(* CODESYS project SmiuUGP_Dubniki.project

Project tree, tasks and I/O mapping:
  CODESYS_Control_for_Raspberry_Pi : CODESYS Control for Raspberry Pi, 3S - Smart Software Solutions GmbH, version 3.5.7.10
    application Application
      libraries: Util, * (System); AlarmManager, * (Intern); Alarm Manager Interfaces, * (Intern); Standard, * (System); VisuDialogs, * (System)
      task MainTask (cyclic, interval t#50ms, priority 2, watchdog t#1000ms x 1) calls PLC_PRG, GPIO_HANDLER, AlarmChecker
      task VISU_TASK (cyclic, interval 100 ms, priority 30) calls VisuElems.Visu_Prg
      task AlarmManagerTask (cyclic, interval 50 ms, priority 31) calls AlarmManager.Alarm_Prg
      task BusTask (cyclic, interval t#20ms, priority 1, watchdog t#1000ms x 1) calls BusReinit
      program PLC_PRG [ST]
      image pool ImagePool
      program GPIO_HANDLER [ST]
      visualization/
        visualisation monitoring
        ups_s2/
          visualisation ups_s2_state
          visualisation ups_s2_params
        visualisation main
        visualisation info
        visualisation climate
        visualisation alarm
        visualisation schrps
        visualisation shasn
        visualisation logs
        visualisation schrpa
        ups_s1/
          visualisation ups_s1_params
          visualisation ups_s1_state
        ups_a1/
          visualisation ups_a1_params
          visualisation ups_a1_state
        ups_a2/
          visualisation ups_a2_params
          visualisation ups_a2_state
        visualisation climate_log
        visualisation more
      Alarm Configuration
        alarm class Error (priority 10, acknowledge REP)
        alarm class Warning (priority 30, acknowledge REP)
        alarm class Info (priority 100, acknowledge REP)
        AlarmStorage
        text list AlarmGroup
        alarm group AlarmGroup
            1 [Error]: Comparison Equal, ExpressionToCompare TRUE, Expression AlarmChecker.shrpa_in_2_alarm - "Отсутствует напряжение на резервном вводе ЩРПА"
            2 [Error]: Comparison Equal, ExpressionToCompare FALSE, Expression GPIO_HANDLER.IN_4 - "Отсутствует напряжение на основном вводе ШАСН"
            3 [Error]: Comparison Equal, ExpressionToCompare FALSE, Expression GPIO_HANDLER.IN_5 - "Отсутствует напряжение на резервном вводе ШАСН"
            4 [Error]: Comparison Equal, ExpressionToCompare FALSE, Expression PLC_PRG.shrps_ups_bus_1 - "Отсутствует напряжение на ГП 1 ЩРПС"
            5 [Error]: Comparison Equal, ExpressionToCompare FALSE, Expression PLC_PRG.shrps_ups_bus_2 - "Отсутствует напряжение на ГП 2 ЩРПС"
            96 [Error]: Comparison Equal, ExpressionToCompare TRUE, Expression GPIO_HANDLER.IN_2 - "Пожар"
            92 [Error]: Comparison Equal, ExpressionToCompare TRUE, Expression AlarmChecker.ups_s1_out_v_alarm - "Отсутствует напряжение на выходе ИБП С1"
            45 [Error]: Comparison Equal, ExpressionToCompare TRUE, Expression PLC_PRG.mpx_a1_1_alarm - "Авария ИБП А1"
            53 [Error]: Comparison Equal, ExpressionToCompare TRUE, Expression PLC_PRG.mpx_s2_1_alarm - "Авария ИБП С2"
            49 [Error]: Comparison Equal, ExpressionToCompare TRUE, Expression PLC_PRG.mpx_s1_1_alarm - "Авария ИБП С1"
            6 [Error]: Comparison Equal, ExpressionToCompare FALSE, Expression GPIO_HANDLER.IN_6 - "Отсутствует напряжение на шине БП ШАСН"
            97 [Error]: Comparison Equal, ExpressionToCompare TRUE, Expression GPIO_HANDLER.IN_1 - "Нарушение ШОС"
            93 [Error]: Comparison Equal, ExpressionToCompare TRUE, Expression AlarmChecker.ups_s2_out_v_alarm - "Отсутствует напряжение на выходе ИБП С2"
            101 [Error]: Comparison Equal, ExpressionToCompare TRUE, Expression AlarmChecker.shrps_in_2_alarm - "Отсутствует напряжение на резервном вводе ЩРПС"
            0 [Error]: Comparison Equal, ExpressionToCompare TRUE, Expression AlarmChecker.shrpa_in_1_alarm - "Отсутствует напряжение на основном вводе ЩРПА"
            47 [Error]: Comparison Equal, ExpressionToCompare TRUE, Expression PLC_PRG.mpx_a2_1_alarm - "Авария ИБП А2"
            94 [Error]: Comparison Equal, ExpressionToCompare TRUE, Expression AlarmChecker.ups_a1_out_v_alarm - "Отсутствует напряжение на выходе ИБП А1"
            90 [Error]: Comparison Equal, ExpressionToCompare TRUE, Expression AlarmChecker.ups_a1_in_v_alarm - "Отсутствует напряжение на входе ИБП А1"
            88 [Error]: Comparison Equal, ExpressionToCompare TRUE, Expression AlarmChecker.ups_s1_in_v_alarm - "Отсутствует напряжение на входе ИБП С1"
            98 [Error]: Comparison Equal, ExpressionToCompare TRUE, Expression GPIO_HANDLER.IN_3 - "Авария ШОС"
            100 [Error]: Comparison Equal, ExpressionToCompare TRUE, Expression AlarmChecker.shrps_in_1_alarm - "Отсутствует напряжение на основном вводе ЩРПC"
            89 [Error]: Comparison Equal, ExpressionToCompare TRUE, Expression AlarmChecker.ups_s2_in_v_alarm - "Отсутствует напряжение на входе ИБП С2"
            95 [Error]: Comparison Equal, ExpressionToCompare TRUE, Expression AlarmChecker.ups_a2_out_v_alarm - "Отсутствует напряжение на выходе ИБП А2"
            91 [Error]: Comparison Equal, ExpressionToCompare TRUE, Expression AlarmChecker.ups_a2_in_v_alarm - "Отсутствует напряжение на входе ИБП А2"
            7 [Error]: Comparison Equal, ExpressionToCompare FALSE, Expression GPIO_HANDLER.IN_7 - "Отсутствует напряжение на шине ГП ШАСН"
            99 [Error]: Comparison Equal, ExpressionToCompare TRUE, Expression AlarmChecker.shrpa_out_alarm - "Отсутствует напряжение на ШБПА  ЩРПА"
        text list ClimateGroup
        alarm group ClimateGroup
            1 [Info]: Comparison Equal, ExpressionToCompare TRUE, Expression PLC_PRG.climate_auto_state - "Автоматика включена"
            2 [Info]: Comparison Equal, ExpressionToCompare FALSE, Expression PLC_PRG.climate_heat_state - "Обогрев выключен"
            3 [Info]: Comparison Equal, ExpressionToCompare FALSE, Expression PLC_PRG.climate_auto_state - "Автоматика выключена"
            4 [Info]: Comparison Equal, ExpressionToCompare TRUE, Expression PLC_PRG.climate_zaslonka_state - "Заслонка открыта"
            5 [Info]: Comparison Equal, ExpressionToCompare FALSE, Expression PLC_PRG.climate_zaslonka_state - "Заслонка закрыта"
            11 [Info]: Comparison Equal, ExpressionToCompare FALSE, Expression PLC_PRG.climate_heat_door_state - "Обогрев дверей выключен"
            7 [Info]: Comparison Equal, ExpressionToCompare FALSE, Expression PLC_PRG.climate_vent_1_state - "Вентиляторы выключены"
            6 [Info]: Comparison Equal, ExpressionToCompare TRUE, Expression PLC_PRG.climate_vent_1_state - "Вентиляторы включены"
            12 [Info]: Comparison Equal, ExpressionToCompare TRUE, Expression PLC_PRG.climate_temp_low - "Низкая температура"
            13 [Info]: Comparison Equal, ExpressionToCompare TRUE, Expression PLC_PRG.climate_temp_hight - "Высокая температура"
            8 [Info]: Comparison Equal, ExpressionToCompare TRUE, Expression PLC_PRG.climate_condition_1_state - "Кондиционеры включены"
            9 [Info]: Comparison Equal, ExpressionToCompare FALSE, Expression PLC_PRG.climate_condition_1_state - "Кондиционеры выключены"
            10 [Info]: Comparison Equal, ExpressionToCompare TRUE, Expression PLC_PRG.climate_heat_door_state - "Обогрев дверей включен"
            0 [Info]: Comparison Equal, ExpressionToCompare TRUE, Expression PLC_PRG.climate_heat_state - "Обогрев включен"
      program BusReinit [ST]
      program AlarmChecker [ST]
    SoftMotion General Axis Pool
    GPIOs_B_Pi2 : GPIOs B+/Pi2, 3S - Smart Software Solutions GmbH, version 1.1.1.10
        input  Application.GPIO_HANDLER.RAW_IN_10 : BOOL  // digital inputs (GPIO0..GPIO31).Bit5
        input  Application.GPIO_HANDLER.RAW_IN_12 : BOOL  // digital inputs (GPIO0..GPIO31).Bit6
        input  Application.GPIO_HANDLER.RAW_IN_9 : BOOL  // digital inputs (GPIO0..GPIO31).Bit7
        input  Application.GPIO_HANDLER.RAW_IN_8 : BOOL  // digital inputs (GPIO0..GPIO31).Bit8
        input  Application.GPIO_HANDLER.RAW_IN_3 : BOOL  // digital inputs (GPIO0..GPIO31).Bit10
        input  Application.GPIO_HANDLER.RAW_IN_11 : BOOL  // digital inputs (GPIO0..GPIO31).Bit12
        input  Application.GPIO_HANDLER.RAW_IN_1 : BOOL  // digital inputs (GPIO0..GPIO31).Bit13
        input  Application.GPIO_HANDLER.RAW_IN_6 : BOOL  // digital inputs (GPIO0..GPIO31).Bit18
        input  Application.GPIO_HANDLER.RAW_IN_7 : BOOL  // digital inputs (GPIO0..GPIO31).Bit21
        input  Application.GPIO_HANDLER.RAW_IN_5 : BOOL  // digital inputs (GPIO0..GPIO31).Bit23
        input  Application.GPIO_HANDLER.RAW_IN_4 : BOOL  // digital inputs (GPIO0..GPIO31).Bit24
        input  Application.GPIO_HANDLER.RAW_IN_2 : BOOL  // digital inputs (GPIO0..GPIO31).Bit25
        unmapped channels: digital inputs (GPIO0..GPIO31), digital outputs (GPIO0..GPIO31)
    Camera device
      <Empty>
    I²C
    SPI
    Onewire
    Ethernet : Ethernet, 3S - Smart Software Solutions GmbH, version 3.4.2.0
        settings: IPAddress = [192,168,10,200]; SubnetMask = [255,255,255,0]; GatewayAddress = [0,0,0,0]; NetworkInterfaceName = 'eth0'; NetworkInterfaceName = "eth0"
      Modbus_TCP_Master : Modbus TCP Master, 3S - Smart Software Solutions GmbH, version 3.5.4.0
          settings: AutoReconnect = TRUE
        IPS_2_2 : Modbus TCP Slave, 3S - Smart Software Solutions GmbH, version 3.5.4.0
            settings: Unit-ID = 1; ResponseTimeout = 1500; IPAddress = [192, 168, 10, 204]; Input_group.Function Code = 3; Input_group.Read Offset = 16#006D; Input_group.Read Length = 4; Input_group.Write Offset = 0; Input_group.Write Length = 0; Input_group.Cycle Time = 300; Output_group.Function Code = 3; Output_group.Read Offset = 16#0077; Output_group.Read Length = 7; Output_group.Write Offset = 0; Output_group.Write Length = 0; Output_group.Cycle Time = 300; Bypass_group.Function Code = 3; Bypass_group.Read Offset = 16#0081; Bypass_group.Read Length = 4; Bypass_group.Write Offset = 0; Bypass_group.Write Length = 0; Bypass_group.Cycle Time = 300; Battarey_group.Function Code = 3; Battarey_group.Read Offset = 16#0063; Battarey_group.Read Length = 4; Battarey_group.Write Offset = 0; Battarey_group.Write Length = 0; Battarey_group.Cycle Time = 300; Inv_Byp.Function Code = 3; Inv_Byp.Read Offset = 16#0095; Inv_Byp.Read Length = 1; Inv_Byp.Write Offset = 0; Inv_Byp.Write Length = 0; Inv_Byp.Cycle Time = 300; Status_group2.Function Code = 3; Status_group2.Read Offset = 16#0031; Status_group2.Read Length = 4; Status_group2.Write Offset = 0; Status_group2.Write Length = 0; Status_group2.Cycle Time = 300; Ivertor.Function Code = 3;
              Ivertor.Read Offset = 16#0096; Ivertor.Read Length = 1; Ivertor.Write Offset = 0; Ivertor.Write Length = 0; Ivertor.Cycle Time = 300; Battarey_temp.Function Code = 3; Battarey_temp.Read Offset = 16#001D; Battarey_temp.Read Length = 1; Battarey_temp.Write Offset = 0; Battarey_temp.Write Length = 0; Battarey_temp.Cycle Time = 300; Fault_grup.Function Code = 3; Fault_grup.Read Offset = 16#009F; Fault_grup.Read Length = 7; Fault_grup.Write Offset = 0; Fault_grup.Write Length = 0; Fault_grup.Cycle Time = 300
            input  Application.PLC_PRG.mpx_s2_1_in_freq : WORD  // Input_group.Input_group
            input  Application.PLC_PRG.mpx_s2_1_in_v_1 : WORD  // Input_group.Input_group
            input  Application.PLC_PRG.mpx_s2_1_in_v_2 : WORD  // Input_group.Input_group
            input  Application.PLC_PRG.mpx_s2_1_in_v_3 : WORD  // Input_group.Input_group
            input  Application.PLC_PRG.mpx_s2_1_output_freq : WORD  // Output_group.Output_group
            input  Application.PLC_PRG.mpx_s2_1_output_v_1 : WORD  // Output_group.Output_group
            input  Application.PLC_PRG.mpx_s2_1_output_v_2 : WORD  // Output_group.Output_group
            input  Application.PLC_PRG.mpx_s2_1_output_v_3 : WORD  // Output_group.Output_group
            input  Application.PLC_PRG.mpx_s2_1_load_ph_1 : WORD  // Output_group.Output_group
            input  Application.PLC_PRG.mpx_s2_1_load_ph_2 : WORD  // Output_group.Output_group
            input  Application.PLC_PRG.mpx_s2_1_load_ph_3 : WORD  // Output_group.Output_group
            input  Application.PLC_PRG.mpx_s2_1_bypass_freq : WORD  // Bypass_group.Bypass_group
            input  Application.PLC_PRG.mpx_s2_1_bypass_v_1 : WORD  // Bypass_group.Bypass_group
            input  Application.PLC_PRG.mpx_s2_1_bypass_v_2 : WORD  // Bypass_group.Bypass_group
            input  Application.PLC_PRG.mpx_s2_1_bypass_v_3 : WORD  // Bypass_group.Bypass_group
            input  Application.PLC_PRG.mpx_s2_1_battery_voltage : WORD  // Battarey_group.Battarey_group
            input  Application.PLC_PRG.mpx_s2_1_battery_capacity : WORD  // Battarey_group.Battarey_group
            input  Application.PLC_PRG.mpx_s2_time_m : WORD  // Battarey_group.Battarey_group
            input  Application.PLC_PRG.mpx_s2_1_battery_current : WORD  // Battarey_group.Battarey_group
            input  Application.PLC_PRG.mpx_s2_1_inv_byp : ARRAY[0..0] OF WORD  // Inv_Byp
            input  Application.PLC_PRG.mpx_s2_1_state_reg : WORD  // Status_group2.Status_group2
            input  Application.PLC_PRG.mpx_s2_1_Invertor : ARRAY[0..0] OF WORD  // Ivertor
            input  Application.PLC_PRG.mpx_s2_1_temp : ARRAY[0..0] OF WORD  // Battarey_temp
            input  Application.PLC_PRG.mpx_s2_1_emergency : WORD  // Fault_grup.Fault_grup
            input  Application.PLC_PRG.mpx_s2_1_overload : WORD  // Fault_grup.Fault_grup
            input  Application.PLC_PRG.mpx_s2_1_outfail : WORD  // Fault_grup.Fault_grup
            input  Application.PLC_PRG.mpx_s2_1_overtemp : WORD  // Fault_grup.Fault_grup
            unmapped channels: Input_group, Output_group, Bypass_group, Battarey_group, Status_group2, Fault_grup
        IPS_2_1 : Modbus TCP Slave, 3S - Smart Software Solutions GmbH, version 3.5.4.0
            settings: Unit-ID = 1; ResponseTimeout = 1500; IPAddress = [192, 168, 10, 203]; Input_group.Function Code = 3; Input_group.Read Offset = 16#006D; Input_group.Read Length = 4; Input_group.Write Offset = 0; Input_group.Write Length = 0; Input_group.Cycle Time = 300; Output_group.Function Code = 3; Output_group.Read Offset = 16#0077; Output_group.Read Length = 7; Output_group.Write Offset = 0; Output_group.Write Length = 0; Output_group.Cycle Time = 300; Bypass_group.Function Code = 3; Bypass_group.Read Offset = 16#0081; Bypass_group.Read Length = 4; Bypass_group.Write Offset = 0; Bypass_group.Write Length = 0; Bypass_group.Cycle Time = 300; Battarey_group.Function Code = 3; Battarey_group.Read Offset = 16#0063; Battarey_group.Read Length = 4; Battarey_group.Write Offset = 0; Battarey_group.Write Length = 0; Battarey_group.Cycle Time = 300; Status2_group.Function Code = 3; Status2_group.Read Offset = 16#0031; Status2_group.Read Length = 4; Status2_group.Write Offset = 0; Status2_group.Write Length = 0; Status2_group.Cycle Time = 300; Invertor.Function Code = 3; Invertor.Read Offset = 16#0096; Invertor.Read Length = 1; Invertor.Write Offset = 0; Invertor.Write Length = 0; Invertor.Cycle Time = 300; Battarey_temp.Function Code = 3;
              Battarey_temp.Read Offset = 16#001D; Battarey_temp.Read Length = 1; Battarey_temp.Write Offset = 0; Battarey_temp.Write Length = 0; Battarey_temp.Cycle Time = 300; Inv_Byp.Function Code = 3; Inv_Byp.Read Offset = 16#0095; Inv_Byp.Read Length = 1; Inv_Byp.Write Offset = 0; Inv_Byp.Write Length = 0; Inv_Byp.Cycle Time = 300; Fault_group.Function Code = 3; Fault_group.Read Offset = 16#009F; Fault_group.Read Length = 7; Fault_group.Write Offset = 0; Fault_group.Write Length = 0; Fault_group.Cycle Time = 300
            input  Application.PLC_PRG.mpx_s1_1_in_freq : WORD  // Input_group.Input_group
            input  Application.PLC_PRG.mpx_s1_1_in_v_1 : WORD  // Input_group.Input_group
            input  Application.PLC_PRG.mpx_s1_1_in_v_2 : WORD  // Input_group.Input_group
            input  Application.PLC_PRG.mpx_s1_1_in_v_3 : WORD  // Input_group.Input_group
            input  Application.PLC_PRG.mpx_s1_1_output_freq : WORD  // Output_group.Output_group
            input  Application.PLC_PRG.mpx_s1_1_output_v_1 : WORD  // Output_group.Output_group
            input  Application.PLC_PRG.mpx_s1_1_output_v_2 : WORD  // Output_group.Output_group
            input  Application.PLC_PRG.mpx_s1_1_output_v_3 : WORD  // Output_group.Output_group
            input  Application.PLC_PRG.mpx_s1_1_load_ph_1 : WORD  // Output_group.Output_group
            input  Application.PLC_PRG.mpx_s1_1_load_ph_2 : WORD  // Output_group.Output_group
            input  Application.PLC_PRG.mpx_s1_1_load_ph_3 : WORD  // Output_group.Output_group
            input  Application.PLC_PRG.mpx_s1_1_bypass_freq : WORD  // Bypass_group.Bypass_group
            input  Application.PLC_PRG.mpx_s1_1_bypass_v_1 : WORD  // Bypass_group.Bypass_group
            input  Application.PLC_PRG.mpx_s1_1_bypass_v_2 : WORD  // Bypass_group.Bypass_group
            input  Application.PLC_PRG.mpx_s1_1_bypass_v_3 : WORD  // Bypass_group.Bypass_group
            input  Application.PLC_PRG.mpx_s1_1_battery_voltage : WORD  // Battarey_group.Battarey_group
            input  Application.PLC_PRG.mpx_s1_1_battery_capacity : WORD  // Battarey_group.Battarey_group
            input  Application.PLC_PRG.mpx_s1_time_m : WORD  // Battarey_group.Battarey_group
            input  Application.PLC_PRG.mpx_s1_1_battery_current : WORD  // Battarey_group.Battarey_group
            input  Application.PLC_PRG.mpx_s1_1_state_reg : WORD  // Status2_group.Status2_group
            input  Application.PLC_PRG.mpx_s1_1_Invertor : ARRAY[0..0] OF WORD  // Invertor
            input  Application.PLC_PRG.mpx_s1_1_temp : ARRAY[0..0] OF WORD  // Battarey_temp
            input  Application.PLC_PRG.mpx_s1_1_inv_byp : ARRAY[0..0] OF WORD  // Inv_Byp
            input  Application.PLC_PRG.mpx_s1_1_emergency : WORD  // Fault_group.Fault_group
            input  Application.PLC_PRG.mpx_s1_1_overload : WORD  // Fault_group.Fault_group
            input  Application.PLC_PRG.mpx_s1_1_outfail : WORD  // Fault_group.Fault_group
            input  Application.PLC_PRG.mpx_s1_1_overtemp : WORD  // Fault_group.Fault_group
            unmapped channels: Input_group, Output_group, Bypass_group, Battarey_group, Status2_group, Fault_group
        IPS_1_1 : Modbus TCP Slave, 3S - Smart Software Solutions GmbH, version 3.5.4.0
            settings: Unit-ID = 1; ResponseTimeout = 1500; IPAddress = [192, 168, 10, 201]; Input_group.Function Code = 3; Input_group.Read Offset = 16#006D; Input_group.Read Length = 4; Input_group.Write Offset = 0; Input_group.Write Length = 0; Input_group.Cycle Time = 300; Output_group.Function Code = 3; Output_group.Read Offset = 16#0077; Output_group.Read Length = 5; Output_group.Write Offset = 0; Output_group.Write Length = 0; Output_group.Cycle Time = 300; Bypass_group.Function Code = 3; Bypass_group.Read Offset = 16#0081; Bypass_group.Read Length = 2; Bypass_group.Write Offset = 0; Bypass_group.Write Length = 0; Bypass_group.Cycle Time = 300; Battarey_group.Function Code = 3; Battarey_group.Read Offset = 16#0063; Battarey_group.Read Length = 4; Battarey_group.Write Offset = 0; Battarey_group.Write Length = 0; Battarey_group.Cycle Time = 300; Status_group2.Function Code = 3; Status_group2.Read Offset = 16#0031; Status_group2.Read Length = 4; Status_group2.Write Offset = 0; Status_group2.Write Length = 0; Status_group2.Cycle Time = 300; Invertor.Function Code = 3; Invertor.Read Offset = 16#0096; Invertor.Read Length = 1; Invertor.Write Offset = 0; Invertor.Write Length = 0; Invertor.Cycle Time = 300; Battarey_temp.Function Code = 3;
              Battarey_temp.Read Offset = 16#001D; Battarey_temp.Read Length = 1; Battarey_temp.Write Offset = 0; Battarey_temp.Write Length = 0; Battarey_temp.Cycle Time = 300; Inv_Byp.Function Code = 3; Inv_Byp.Read Offset = 16#0095; Inv_Byp.Read Length = 1; Inv_Byp.Write Offset = 0; Inv_Byp.Write Length = 0; Inv_Byp.Cycle Time = 300; Fault_group.Function Code = 3; Fault_group.Read Offset = 16#009F; Fault_group.Read Length = 7; Fault_group.Write Offset = 0; Fault_group.Write Length = 0; Fault_group.Cycle Time = 300
            input  Application.PLC_PRG.mpx_a1_1_in_freq : WORD  // Input_group.Input_group
            input  Application.PLC_PRG.mpx_a1_1_in_v_1 : WORD  // Input_group.Input_group
            input  Application.PLC_PRG.mpx_a1_1_in_v_2 : WORD  // Input_group.Input_group
            input  Application.PLC_PRG.mpx_a1_1_in_v_3 : WORD  // Input_group.Input_group
            input  Application.PLC_PRG.mpx_a1_1_output_freq : WORD  // Output_group.Output_group
            input  Application.PLC_PRG.mpx_a1_1_output_v_1 : WORD  // Output_group.Output_group
            input  Application.PLC_PRG.mpx_a1_1_load_ph_1 : WORD  // Output_group.Output_group
            input  Application.PLC_PRG.mpx_a1_1_bypass_freq : WORD  // Bypass_group.Bypass_group
            input  Application.PLC_PRG.mpx_a1_1_bypass_v_1 : WORD  // Bypass_group.Bypass_group
            input  Application.PLC_PRG.mpx_a1_1_battery_voltage : WORD  // Battarey_group.Battarey_group
            input  Application.PLC_PRG.mpx_a1_1_battery_capacity : WORD  // Battarey_group.Battarey_group
            input  Application.PLC_PRG.mpx_a1_time_m : WORD  // Battarey_group.Battarey_group
            input  Application.PLC_PRG.mpx_a1_1_battery_current : WORD  // Battarey_group.Battarey_group
            input  Application.PLC_PRG.mpx_a1_1_state_reg : WORD  // Status_group2.Status_group2
            input  Application.PLC_PRG.mpx_a1_1_Invertor : ARRAY[0..0] OF WORD  // Invertor
            input  Application.PLC_PRG.mpx_a1_1_temp : ARRAY[0..0] OF WORD  // Battarey_temp
            input  Application.PLC_PRG.mpx_a1_1_inv_byp : ARRAY[0..0] OF WORD  // Inv_Byp
            input  Application.PLC_PRG.mpx_a1_1_emergency : WORD  // Fault_group.Fault_group
            input  Application.PLC_PRG.mpx_a1_1_overload : WORD  // Fault_group.Fault_group
            input  Application.PLC_PRG.mpx_a1_1_outfail : WORD  // Fault_group.Fault_group
            input  Application.PLC_PRG.mpx_a1_1_overtemp : WORD  // Fault_group.Fault_group
            unmapped channels: Input_group, Output_group, Bypass_group, Battarey_group, Status_group2, Fault_group
        IPS_1_2 : Modbus TCP Slave, 3S - Smart Software Solutions GmbH, version 3.5.4.0
            settings: Unit-ID = 1; ResponseTimeout = 1500; IPAddress = [192, 168, 10, 202]; Input_group.Function Code = 3; Input_group.Read Offset = 16#006D; Input_group.Read Length = 4; Input_group.Write Offset = 0; Input_group.Write Length = 0; Input_group.Cycle Time = 300; Output_group.Function Code = 3; Output_group.Read Offset = 16#0077; Output_group.Read Length = 5; Output_group.Write Offset = 0; Output_group.Write Length = 0; Output_group.Cycle Time = 300; Bypass_group.Function Code = 3; Bypass_group.Read Offset = 16#0081; Bypass_group.Read Length = 2; Bypass_group.Write Offset = 0; Bypass_group.Write Length = 0; Bypass_group.Cycle Time = 300; Battarey_group.Function Code = 3; Battarey_group.Read Offset = 16#0063; Battarey_group.Read Length = 4; Battarey_group.Write Offset = 0; Battarey_group.Write Length = 0; Battarey_group.Cycle Time = 300; Status_group2.Function Code = 3; Status_group2.Read Offset = 16#0031; Status_group2.Read Length = 4; Status_group2.Write Offset = 0; Status_group2.Write Length = 0; Status_group2.Cycle Time = 300; Invertor.Function Code = 3; Invertor.Read Offset = 16#0096; Invertor.Read Length = 1; Invertor.Write Offset = 0; Invertor.Write Length = 0; Invertor.Cycle Time = 300; Battarey_temp.Function Code = 3;
              Battarey_temp.Read Offset = 16#001D; Battarey_temp.Read Length = 1; Battarey_temp.Write Offset = 0; Battarey_temp.Write Length = 0; Battarey_temp.Cycle Time = 300; Inv_Byp.Function Code = 3; Inv_Byp.Read Offset = 16#0095; Inv_Byp.Read Length = 1; Inv_Byp.Write Offset = 0; Inv_Byp.Write Length = 0; Inv_Byp.Cycle Time = 300; Fault_group.Function Code = 3; Fault_group.Read Offset = 16#009F; Fault_group.Read Length = 7; Fault_group.Write Offset = 0; Fault_group.Write Length = 0; Fault_group.Cycle Time = 300
            input  Application.PLC_PRG.mpx_a2_1_in_freq : WORD  // Input_group.Input_group
            input  Application.PLC_PRG.mpx_a2_1_in_v_1 : WORD  // Input_group.Input_group
            input  Application.PLC_PRG.mpx_a2_1_in_v_2 : WORD  // Input_group.Input_group
            input  Application.PLC_PRG.mpx_a2_1_in_v_3 : WORD  // Input_group.Input_group
            input  Application.PLC_PRG.mpx_a2_1_output_freq : WORD  // Output_group.Output_group
            input  Application.PLC_PRG.mpx_a2_1_output_v_1 : WORD  // Output_group.Output_group
            input  Application.PLC_PRG.mpx_a2_1_load_ph_1 : WORD  // Output_group.Output_group
            input  Application.PLC_PRG.mpx_a2_1_bypass_freq : WORD  // Bypass_group.Bypass_group
            input  Application.PLC_PRG.mpx_a2_1_bypass_v_1 : WORD  // Bypass_group.Bypass_group
            input  Application.PLC_PRG.mpx_a2_1_battery_voltage : WORD  // Battarey_group.Battarey_group
            input  Application.PLC_PRG.mpx_a2_1_battery_capacity : WORD  // Battarey_group.Battarey_group
            input  Application.PLC_PRG.mpx_a2_time_m : WORD  // Battarey_group.Battarey_group
            input  Application.PLC_PRG.mpx_a2_1_battery_current : WORD  // Battarey_group.Battarey_group
            input  Application.PLC_PRG.mpx_a2_1_state_reg : WORD  // Status_group2.Status_group2
            input  Application.PLC_PRG.mpx_a2_1_Invertor : ARRAY[0..0] OF WORD  // Invertor
            input  Application.PLC_PRG.mpx_a2_1_temp : ARRAY[0..0] OF WORD  // Battarey_temp
            input  Application.PLC_PRG.mpx_a2_1_inv_byp : ARRAY[0..0] OF WORD  // Inv_Byp
            input  Application.PLC_PRG.mpx_a2_1_emergency : WORD  // Fault_group.Fault_group
            input  Application.PLC_PRG.mpx_a2_1_overload : WORD  // Fault_group.Fault_group
            input  Application.PLC_PRG.mpx_a2_1_outfail : WORD  // Fault_group.Fault_group
            input  Application.PLC_PRG.mpx_a2_1_overtemp : WORD  // Fault_group.Fault_group
            unmapped channels: Input_group, Output_group, Bypass_group, Battarey_group, Status_group2, Fault_group
    ModbusIN : Modbus COM, 3S - Smart Software Solutions GmbH, version 3.4.0.0
        settings: DataBits = 8; StopBits = 1; ComPort = 1
      ModbusMaster : Modbus Master, COM Port, 3S - Smart Software Solutions GmbH, version 3.5.5.0
          settings: Transmission = 'RTU'; ResponseTimeout = 60; TimeBetweenFrames = 20; Auto-restart communication = TRUE
        PLC : Modbus Slave, COM Port, 3S - Smart Software Solutions GmbH, version 3.5.4.0
            settings: SlaveAddress = 1; ResponseTimeout = 100; UseExtendedFunctionCodes = TRUE; Channel 0.Function Code = 3; Channel 0.Read Offset = 16#EB28; Channel 0.Read Length = 3; Channel 0.Write Offset = 0; Channel 0.Write Length = 0; Channel 0.Cycle Time = 500
            input  Application.PLC_PRG.climate_temp_in : WORD  // Channel 0.Channel 0
            input  Application.PLC_PRG.climate_temp_out : WORD  // Channel 0.Channel 0
            input  Application.PLC_PRG.climate_state_reg : WORD  // Channel 0.Channel 0
            unmapped channels: Channel 0
        SHRPA_ICP_CON : Modbus Slave, COM Port, 3S - Smart Software Solutions GmbH, version 3.5.4.0
            settings: SlaveAddress = 101; ResponseTimeout = 50; UseExtendedFunctionCodes = TRUE; DI.Function Code = 2; DI.Read Offset = 16#0000; DI.Read Length = 16; DI.Write Offset = 0; DI.Write Length = 0; DI.Cycle Time = 100
            input  Application.PLC_PRG.shrpa_in_1 : BOOL  // DI.DI.Bit0
            input  Application.PLC_PRG.shrpa_in_2 : BOOL  // DI.DI.Bit1
            input  Application.PLC_PRG.shrpa_ups_in_1_raw : BOOL  // DI.DI.Bit2
            input  Application.PLC_PRG.shrpa_ups_in_2_raw : BOOL  // DI.DI.Bit3
            input  Application.PLC_PRG.shrpa_input_switch_state_1 : BOOL  // DI.DI.Bit4
            input  Application.PLC_PRG.shrpa_input_switch_state_2 : BOOL  // DI.DI.Bit5
            input  Application.PLC_PRG.shrpa_ups_out_1 : BOOL  // DI.DI.Bit6
            input  Application.PLC_PRG.shrpa_ups_out_2 : BOOL  // DI.DI.Bit7
            input  Application.PLC_PRG.shrpa_load_line_1_source_state_1 : BOOL  // DI.DI.Bit0
            input  Application.PLC_PRG.shrpa_load_line_1_source_state_2 : BOOL  // DI.DI.Bit1
            input  Application.PLC_PRG.shrpa_load_line_2_source_state_2 : BOOL  // DI.DI.Bit2
            input  Application.PLC_PRG.shrpa_load_line_2_source_state_1 : BOOL  // DI.DI.Bit3
            input  Application.PLC_PRG.shrpa_input_tv1 : BOOL  // DI.DI.Bit4
            input  Application.PLC_PRG.shrpa_bypass_in_1 : BOOL  // DI.DI.Bit5
            input  Application.PLC_PRG.shrpa_bypass_in_2 : BOOL  // DI.DI.Bit6
            unmapped channels: DI
        SHRPS_ICP_CON : Modbus Slave, COM Port, 3S - Smart Software Solutions GmbH, version 3.5.4.0
            settings: SlaveAddress = 102; ResponseTimeout = 50; UseExtendedFunctionCodes = TRUE; DI.Function Code = 2; DI.Read Offset = 16#0000; DI.Read Length = 16; DI.Write Offset = 0; DI.Write Length = 0; DI.Cycle Time = 100
            input  Application.PLC_PRG.shrps_in_1 : BOOL  // DI.DI.Bit0
            input  Application.PLC_PRG.shrps_in_2 : BOOL  // DI.DI.Bit1
            input  Application.PLC_PRG.shrps_ups_in_1 : BOOL  // DI.DI.Bit2
            input  Application.PLC_PRG.shrps_bypass_in_1 : BOOL  // DI.DI.Bit3
            input  Application.PLC_PRG.shrps_ups_in_2 : BOOL  // DI.DI.Bit4
            input  Application.PLC_PRG.shrps_bypass_in_2 : BOOL  // DI.DI.Bit5
            input  Application.PLC_PRG.shrps_ups_out_1 : BOOL  // DI.DI.Bit6
            input  Application.PLC_PRG.shrps_ups_out_2 : BOOL  // DI.DI.Bit7
            input  Application.PLC_PRG.shrps_bypass_out : BOOL  // DI.DI.Bit0
            input  Application.PLC_PRG.shrps_ups_bus_1_raw : BOOL  // DI.DI.Bit1
            input  Application.PLC_PRG.shrps_ups_bus_2_raw : BOOL  // DI.DI.Bit2
            unmapped channels: DI
        SHASN_ICP_CON : Modbus Slave, COM Port, 3S - Smart Software Solutions GmbH, version 3.5.4.0
            settings: SlaveAddress = 103; ResponseTimeout = 50; UseExtendedFunctionCodes = TRUE; DI.Function Code = 2; DI.Read Offset = 16#0000; DI.Read Length = 16; DI.Write Offset = 0; DI.Write Length = 0; DI.Cycle Time = 100
            unmapped channels: DI
        SHRPA_ELNET_2 : Modbus Slave, COM Port, 3S - Smart Software Solutions GmbH, version 3.5.4.0
            settings: SlaveAddress = 12; ResponseTimeout = 100; UseExtendedFunctionCodes = TRUE; Voltage.Function Code = 3; Voltage.Read Offset = 16#0001; Voltage.Read Length = 6; Voltage.Write Offset = 0; Voltage.Write Length = 0; Voltage.Cycle Time = 500; Current.Function Code = 3; Current.Read Offset = 16#000D; Current.Read Length = 6; Current.Write Offset = 0; Current.Write Length = 0; Current.Cycle Time = 500
            input  Application.PLC_PRG.shrpa_voltage_registers2 : ARRAY[0..5] OF WORD  // Voltage
            unmapped channels: Current
        SHRPA_ELNET_1 : Modbus Slave, COM Port, 3S - Smart Software Solutions GmbH, version 3.5.4.0
            settings: SlaveAddress = 11; ResponseTimeout = 100; UseExtendedFunctionCodes = TRUE; Voltage.Function Code = 3; Voltage.Read Offset = 16#0001; Voltage.Read Length = 6; Voltage.Write Offset = 0; Voltage.Write Length = 0; Voltage.Cycle Time = 500; Current.Function Code = 3; Current.Read Offset = 16#000D; Current.Read Length = 6; Current.Write Offset = 0; Current.Write Length = 0; Current.Cycle Time = 500
            input  Application.PLC_PRG.shrpa_voltage_registers1 : ARRAY[0..5] OF WORD  // Voltage
            unmapped channels: Current
        SHRPA_ELNET_3 : Modbus Slave, COM Port, 3S - Smart Software Solutions GmbH, version 3.5.4.0
            settings: SlaveAddress = 13; ResponseTimeout = 100; UseExtendedFunctionCodes = TRUE; Voltage.Function Code = 3; Voltage.Read Offset = 16#0001; Voltage.Read Length = 2; Voltage.Write Offset = 0; Voltage.Write Length = 0; Voltage.Cycle Time = 500; Current.Function Code = 3; Current.Read Offset = 16#000D; Current.Read Length = 2; Current.Write Offset = 0; Current.Write Length = 0; Current.Cycle Time = 500; Freq.Function Code = 3; Freq.Read Offset = 16#0033; Freq.Read Length = 2; Freq.Write Offset = 0; Freq.Write Length = 0; Freq.Cycle Time = 500
            input  Application.PLC_PRG.shrpa_voltage_registers3 : ARRAY[0..1] OF WORD  // Voltage
            input  Application.PLC_PRG.shrpa_current_registers3 : ARRAY[0..1] OF WORD  // Current
            input  Application.PLC_PRG.shrpa_freq_registers3 : ARRAY[0..1] OF WORD  // Freq
        SHRPA_ELNET_4 : Modbus Slave, COM Port, 3S - Smart Software Solutions GmbH, version 3.5.4.0
            settings: SlaveAddress = 14; ResponseTimeout = 100; UseExtendedFunctionCodes = TRUE; Voltage.Function Code = 3; Voltage.Read Offset = 16#0001; Voltage.Read Length = 2; Voltage.Write Offset = 0; Voltage.Write Length = 0; Voltage.Cycle Time = 500; Current.Function Code = 3; Current.Read Offset = 16#000D; Current.Read Length = 2; Current.Write Offset = 0; Current.Write Length = 0; Current.Cycle Time = 500; Freq.Function Code = 3; Freq.Read Offset = 16#0033; Freq.Read Length = 2; Freq.Write Offset = 0; Freq.Write Length = 0; Freq.Cycle Time = 500
            input  Application.PLC_PRG.shrpa_voltage_registers4 : ARRAY[0..1] OF WORD  // Voltage
            input  Application.PLC_PRG.shrpa_current_registers4 : ARRAY[0..1] OF WORD  // Current
            input  Application.PLC_PRG.shrpa_freq_registers4 : ARRAY[0..1] OF WORD  // Freq
        SHRPS_ELNET_1 : Modbus Slave, COM Port, 3S - Smart Software Solutions GmbH, version 3.5.4.0
            settings: SlaveAddress = 21; ResponseTimeout = 100; UseExtendedFunctionCodes = TRUE; Voltage.Function Code = 3; Voltage.Read Offset = 16#0001; Voltage.Read Length = 6; Voltage.Write Offset = 0; Voltage.Write Length = 0; Voltage.Cycle Time = 500; Current.Function Code = 3; Current.Read Offset = 16#000D; Current.Read Length = 6; Current.Write Offset = 0; Current.Write Length = 0; Current.Cycle Time = 500
            input  Application.PLC_PRG.shrps_voltage_registers1 : ARRAY[0..5] OF WORD  // Voltage
            unmapped channels: Current
        SHRPS_ELNET_2 : Modbus Slave, COM Port, 3S - Smart Software Solutions GmbH, version 3.5.4.0
            settings: SlaveAddress = 22; ResponseTimeout = 100; UseExtendedFunctionCodes = TRUE; Voltage.Function Code = 3; Voltage.Read Offset = 16#0001; Voltage.Read Length = 6; Voltage.Write Offset = 0; Voltage.Write Length = 0; Voltage.Cycle Time = 500; Current.Function Code = 3; Current.Read Offset = 16#000D; Current.Read Length = 6; Current.Write Offset = 0; Current.Write Length = 0; Current.Cycle Time = 500
            input  Application.PLC_PRG.shrps_voltage_registers2 : ARRAY[0..5] OF WORD  // Voltage
            unmapped channels: Current
        SHRPS_ELNET_3 : Modbus Slave, COM Port, 3S - Smart Software Solutions GmbH, version 3.5.4.0
            settings: SlaveAddress = 23; ResponseTimeout = 100; UseExtendedFunctionCodes = TRUE; Voltage.Function Code = 3; Voltage.Read Offset = 16#0001; Voltage.Read Length = 6; Voltage.Write Offset = 0; Voltage.Write Length = 0; Voltage.Cycle Time = 500; Current.Function Code = 3; Current.Read Offset = 16#000D; Current.Read Length = 6; Current.Write Offset = 0; Current.Write Length = 0; Current.Cycle Time = 500
            input  Application.PLC_PRG.shrps_voltage_registers3 : ARRAY[0..5] OF WORD  // Voltage
            unmapped channels: Current
        SHRPS_ELNET_4 : Modbus Slave, COM Port, 3S - Smart Software Solutions GmbH, version 3.5.4.0
            settings: SlaveAddress = 24; ResponseTimeout = 100; UseExtendedFunctionCodes = TRUE; Voltage.Function Code = 3; Voltage.Read Offset = 16#0001; Voltage.Read Length = 6; Voltage.Write Offset = 0; Voltage.Write Length = 0; Voltage.Cycle Time = 500; Current.Function Code = 3; Current.Read Offset = 16#000D; Current.Read Length = 6; Current.Write Offset = 0; Current.Write Length = 0; Current.Cycle Time = 500
            input  Application.PLC_PRG.shrps_voltage_registers4 : ARRAY[0..5] OF WORD  // Voltage
            unmapped channels: Current
    ModbusOUT : Modbus COM, 3S - Smart Software Solutions GmbH, version 3.4.0.0
        settings: DataBits = 8; StopBits = 1; ComPort = 2
      Modbus_Serial_Device : Modbus Serial Device, 3S - Smart Software Solutions GmbH, version 3.5.5.0
          output Application.PLC_PRG.mpx_s1_1_battery_capacity : WORD  // Outputs.Outputs
          output Application.PLC_PRG.mpx_s1_1_battery_current : WORD  // Outputs.Outputs
          output Application.PLC_PRG.mpx_s1_1_battery_time : WORD  // Outputs.Outputs
          output Application.PLC_PRG.mpx_s1_1_battery_voltage : WORD  // Outputs.Outputs
          output Application.PLC_PRG.mpx_s1_1_bypass_v_1 : WORD  // Outputs.Outputs
          output Application.PLC_PRG.mpx_s1_1_bypass_v_2 : WORD  // Outputs.Outputs
          output Application.PLC_PRG.mpx_s1_1_bypass_v_3 : WORD  // Outputs.Outputs
          output Application.PLC_PRG.mpx_s1_1_in_v_1 : WORD  // Outputs.Outputs
          output Application.PLC_PRG.mpx_s1_1_in_v_2 : WORD  // Outputs.Outputs
          output Application.PLC_PRG.mpx_s1_1_in_v_3 : WORD  // Outputs.Outputs
          output Application.PLC_PRG.mpx_s1_1_load_ph_1 : WORD  // Outputs.Outputs
          output Application.PLC_PRG.mpx_s1_1_load_ph_2 : WORD  // Outputs.Outputs
          output Application.PLC_PRG.mpx_s1_1_load_ph_3 : WORD  // Outputs.Outputs
          output Application.PLC_PRG.mpx_s1_1_output_active_power_1 : WORD  // Outputs.Outputs
          output Application.PLC_PRG.mpx_s1_1_output_active_power_2 : WORD  // Outputs.Outputs
          output Application.PLC_PRG.mpx_s1_1_output_active_power_3 : WORD  // Outputs.Outputs
          output Application.PLC_PRG.mpx_s1_1_output_freq : WORD  // Outputs.Outputs
          output Application.PLC_PRG.mpx_s1_1_output_v_1 : WORD  // Outputs.Outputs
          output Application.PLC_PRG.mpx_s1_1_output_v_2 : WORD  // Outputs.Outputs
          output Application.PLC_PRG.mpx_s1_1_output_v_3 : WORD  // Outputs.Outputs
          output Application.PLC_PRG.mpx_s1_1_temp : WORD  // Outputs.Outputs
          output Application.PLC_PRG.ips2_1_state : WORD  // Outputs.Outputs
          output Application.PLC_PRG.mpx_s2_1_battery_capacity : WORD  // Outputs.Outputs
          output Application.PLC_PRG.mpx_s2_1_battery_current : WORD  // Outputs.Outputs
          output Application.PLC_PRG.mpx_s2_1_battery_time : WORD  // Outputs.Outputs
          output Application.PLC_PRG.mpx_s2_1_battery_voltage : WORD  // Outputs.Outputs
          output Application.PLC_PRG.mpx_s2_1_bypass_v_1 : WORD  // Outputs.Outputs
          output Application.PLC_PRG.mpx_s2_1_bypass_v_2 : WORD  // Outputs.Outputs
          output Application.PLC_PRG.mpx_s2_1_bypass_v_3 : WORD  // Outputs.Outputs
          output Application.PLC_PRG.mpx_s2_1_in_v_1 : WORD  // Outputs.Outputs
          output Application.PLC_PRG.mpx_s2_1_in_v_2 : WORD  // Outputs.Outputs
          output Application.PLC_PRG.mpx_s2_1_in_v_3 : WORD  // Outputs.Outputs
          output Application.PLC_PRG.mpx_s2_1_load_ph_1 : WORD  // Outputs.Outputs
          output Application.PLC_PRG.mpx_s2_1_load_ph_2 : WORD  // Outputs.Outputs
          output Application.PLC_PRG.mpx_s2_1_load_ph_3 : WORD  // Outputs.Outputs
          output Application.PLC_PRG.mpx_s2_1_output_active_power_1 : WORD  // Outputs.Outputs
          output Application.PLC_PRG.mpx_s2_1_output_active_power_2 : WORD  // Outputs.Outputs
          output Application.PLC_PRG.mpx_s2_1_output_active_power_3 : WORD  // Outputs.Outputs
          output Application.PLC_PRG.mpx_s2_1_output_freq : WORD  // Outputs.Outputs
          output Application.PLC_PRG.mpx_s2_1_output_v_1 : WORD  // Outputs.Outputs
          output Application.PLC_PRG.mpx_s2_1_output_v_2 : WORD  // Outputs.Outputs
          output Application.PLC_PRG.mpx_s2_1_output_v_3 : WORD  // Outputs.Outputs
          output Application.PLC_PRG.mpx_s2_1_temp : WORD  // Outputs.Outputs
          output Application.PLC_PRG.ips2_2_state : WORD  // Outputs.Outputs
          output Application.PLC_PRG.mpx_a1_1_battery_capacity : WORD  // Outputs.Outputs
          output Application.PLC_PRG.mpx_a1_1_battery_current : WORD  // Outputs.Outputs
          output Application.PLC_PRG.mpx_a1_1_battery_time : WORD  // Outputs.Outputs
          output Application.PLC_PRG.mpx_a1_1_battery_voltage : WORD  // Outputs.Outputs
          output Application.PLC_PRG.mpx_a1_1_bypass_v_1 : WORD  // Outputs.Outputs
          output Application.PLC_PRG.mpx_a1_1_in_v_1 : WORD  // Outputs.Outputs
          output Application.PLC_PRG.mpx_a1_1_in_v_2 : WORD  // Outputs.Outputs
          output Application.PLC_PRG.mpx_a1_1_in_v_3 : WORD  // Outputs.Outputs
          output Application.PLC_PRG.mpx_a1_1_load_ph_1 : WORD  // Outputs.Outputs
          output Application.PLC_PRG.mpx_a1_1_output_active_power_1 : WORD  // Outputs.Outputs
          output Application.PLC_PRG.mpx_a1_1_output_freq : WORD  // Outputs.Outputs
          output Application.PLC_PRG.mpx_a1_1_output_v_1 : WORD  // Outputs.Outputs
          output Application.PLC_PRG.mpx_a1_1_temp : WORD  // Outputs.Outputs
          output Application.PLC_PRG.ips1_1_state : WORD  // Outputs.Outputs
          output Application.PLC_PRG.mpx_a2_1_battery_capacity : WORD  // Outputs.Outputs
          output Application.PLC_PRG.mpx_a2_1_battery_current : WORD  // Outputs.Outputs
          output Application.PLC_PRG.mpx_a2_1_battery_time : WORD  // Outputs.Outputs
          output Application.PLC_PRG.mpx_a2_1_battery_voltage : WORD  // Outputs.Outputs
          output Application.PLC_PRG.mpx_a2_1_bypass_v_1 : WORD  // Outputs.Outputs
          output Application.PLC_PRG.mpx_a2_1_in_v_1 : WORD  // Outputs.Outputs
          output Application.PLC_PRG.mpx_a2_1_in_v_2 : WORD  // Outputs.Outputs
          output Application.PLC_PRG.mpx_a2_1_in_v_3 : WORD  // Outputs.Outputs
          output Application.PLC_PRG.mpx_a2_1_load_ph_1 : WORD  // Outputs.Outputs
          output Application.PLC_PRG.mpx_a2_1_output_active_power_1 : WORD  // Outputs.Outputs
          output Application.PLC_PRG.mpx_a2_1_output_freq : WORD  // Outputs.Outputs
          output Application.PLC_PRG.mpx_a2_1_output_v_1 : WORD  // Outputs.Outputs
          output Application.PLC_PRG.mpx_a2_1_temp : WORD  // Outputs.Outputs
          output Application.PLC_PRG.ips1_2_state : WORD  // Outputs.Outputs
          output Application.PLC_PRG.climate_state_reg : WORD  // Outputs.Outputs
          output Application.PLC_PRG.climate_temp_in : WORD  // Outputs.Outputs
          output Application.PLC_PRG.climate_temp_out : WORD  // Outputs.Outputs
          unmapped channels: Inputs, Outputs
  text list GlobalTextList
  5ce3da45-db07-42e7-a21c-a00fff4ed8f6|Images\bg_800.png
  5ce3da45-db07-42e7-a21c-a00fff4ed8f6|Images\mpx_state_bg.png
  5ce3da45-db07-42e7-a21c-a00fff4ed8f6|Images\ups\bypass_line_on.png
  5ce3da45-db07-42e7-a21c-a00fff4ed8f6|Images\ups\bypass_line_off.png
  5ce3da45-db07-42e7-a21c-a00fff4ed8f6|Images\ups\battery_arrow_off.png
  5ce3da45-db07-42e7-a21c-a00fff4ed8f6|Images\ups\battery_arrow_on.png
  5ce3da45-db07-42e7-a21c-a00fff4ed8f6|Images\ups\battery_line_off.png
  5ce3da45-db07-42e7-a21c-a00fff4ed8f6|Images\ups\battery_line_on.png
  5ce3da45-db07-42e7-a21c-a00fff4ed8f6|Images\ups\bypass_arrow_off.png
  5ce3da45-db07-42e7-a21c-a00fff4ed8f6|Images\ups\bypass_arrow_on.png
  5ce3da45-db07-42e7-a21c-a00fff4ed8f6|Images\ups\arrow_off.png
  5ce3da45-db07-42e7-a21c-a00fff4ed8f6|Images\ups\arrow_on.png
  5ce3da45-db07-42e7-a21c-a00fff4ed8f6|C:\workspace\SmiuUGP\Images\Proba.png
  5ce3da45-db07-42e7-a21c-a00fff4ed8f6|C:\workspace\SmiuUGP\Images\main_bg.png
  5ce3da45-db07-42e7-a21c-a00fff4ed8f6|C:\workspace\SmiuUGP\Images\bg_800.png
  5ce3da45-db07-42e7-a21c-a00fff4ed8f6|E:\YandexDisk\Скриншоты\ups.png
  5ce3da45-db07-42e7-a21c-a00fff4ed8f6|C:\workspace\SmiuUGP\Images\mpx_state_bg.png
  5ce3da45-db07-42e7-a21c-a00fff4ed8f6|C:\workspace\SmiuUGP\Images\scheme.png
  5ce3da45-db07-42e7-a21c-a00fff4ed8f6|C:\workspace\SmiuUGP\Images\more_info.png
  5ce3da45-db07-42e7-a21c-a00fff4ed8f6|C:\workspace\SmiuUGP\Images\log.png
  5ce3da45-db07-42e7-a21c-a00fff4ed8f6|C:\workspace\SmiuUGP\Images\gpio_1.png
  5ce3da45-db07-42e7-a21c-a00fff4ed8f6|release_images\schrpa.png
  5ce3da45-db07-42e7-a21c-a00fff4ed8f6|C:\workspace\SmiuUGP\Images\volt.png
  5ce3da45-db07-42e7-a21c-a00fff4ed8f6|release_images\shasn.png
  5ce3da45-db07-42e7-a21c-a00fff4ed8f6|C:\workspace\SmiuUGP\Images\battery.png
  5ce3da45-db07-42e7-a21c-a00fff4ed8f6|C:\workspace\SmiuUGP\Images\climate.png
  5ce3da45-db07-42e7-a21c-a00fff4ed8f6|C:\workspace\SmiuUGP\Images\alert.png
  5ce3da45-db07-42e7-a21c-a00fff4ed8f6|C:\workspace\SmiuUGP\Images\automation.png
  5ce3da45-db07-42e7-a21c-a00fff4ed8f6|E:\SmiuLinux\smiu_logo.png
  5ce3da45-db07-42e7-a21c-a00fff4ed8f6|C:\workspace\SmiuUGP\Images\mini_ups.png
  5ce3da45-db07-42e7-a21c-a00fff4ed8f6|release_images\shrpa.png
  5ce3da45-db07-42e7-a21c-a00fff4ed8f6|release_images\schrps.png
*)

// CODESYS_Control_for_Raspberry_Pi/Application/PLC_PRG
PROGRAM PLC_PRG
VAR	
	// Переменные для работы с ICP DAS
	// ЩРПА
	shrpa_in_1 : BOOL;							// ввод 1
	shrpa_in_2 : BOOL;							// ввод 2
	shrpa_ups_in_1_raw : BOOL;					// инвертировано
	shrpa_ups_in_2_raw : BOOL;					// инвертировано	
	shrpa_ups_in_1 : BOOL;						// ввод ИБП А1
	shrpa_ups_in_2 : BOOL;						// ввод ИБП А2
	shrpa_input_switch_state_1 : BOOL;			// QS1 в 1 положениии
	shrpa_input_switch_state_2 : BOOL;			// QS1 во 2 положениии
	shrpa_ups_out_1 : BOOL;						// выход ИБП А1
	shrpa_ups_out_2 : BOOL;						// выход ИБП А2
	shrpa_load_line_1_source_state_1 : BOOL;	//QS2 в 1 положении
	shrpa_load_line_1_source_state_2 : BOOL;	//QS2 во 2 положении
	shrpa_load_line_2_source_state_1 : BOOL;	//QS3 в 1 положении
	shrpa_load_line_2_source_state_2 : BOOL;	//QS3 во 2 положении
	shrpa_input_tv1 : BOOL	;					// ввод от TV1
	shrpa_bypass_in_1 : BOOL;					// ввод байпаса ИБП А1
	shrpa_bypass_in_2 : BOOL;					// ввод байпаса ИБП А2
	
	// ЩРПС
	shrps_in_1 : BOOL;							// ввод 1
	shrps_in_2 : BOOL;							// ввод 2
	shrps_ups_in_1 : BOOL;						// ввод ИБП C1
	shrps_ups_in_2 : BOOL;						// ввод ИБП C2		
	shrps_bypass_in_1 : BOOL;					// ввод байпаса ИБП C1
	shrps_bypass_in_2 : BOOL;					// ввод байпаса ИБП C2
	shrps_ups_out_1 : BOOL;						// выход ИБП C1
	shrps_ups_out_2 : BOOL;						// выход ИБП C2
	shrps_bypass_out : BOOL;					// 
	shrps_ups_bus_1_raw : BOOL;					// инвертировано
	shrps_ups_bus_2_raw : BOOL;					// инвертировано
	shrps_ups_bus_1 : BOOL;						// Наличие напряжения на шине бесперебойного питания 1
	shrps_ups_bus_2 : BOOL;						// Наличие напряжения на шине бесперебойного питания 2
	
	// Переменные для работы с ElNet LTE
	delay_timeout 			: TIME := T#5S;
	// ЩРПА
	shrpa_voltage_registers1: ARRAY [1..6] OF WORD;
	shrpa_voltage_registers2: ARRAY [1..6] OF WORD;
	shrpa_voltage_registers3: ARRAY [1..2] OF WORD;
	shrpa_voltage_registers4: ARRAY [1..2] OF WORD;
	
	shrpa_current_registers3: ARRAY [1..2] OF WORD;
	shrpa_current_registers4: ARRAY [1..2] OF WORD;
	
	shrpa_freq_registers3: ARRAY [1..2] OF WORD;
	shrpa_freq_registers4: ARRAY [1..2] OF WORD;
	
	Shrpa_voltage_1_delay_timer	: TON;
	Shrpa_voltage_2_delay_timer	: TON;
	Shrpa_voltage_3_delay_timer	: TON;
	Shrpa_voltage_4_delay_timer	: TON;
	
	shrpa_voltage_1_sum_checker : REAL;
	shrpa_voltage_2_sum_checker : REAL;
	
	shrpa_voltage_1_line_1 : REAL;	
	shrpa_voltage_1_line_2 : REAL;	
	shrpa_voltage_1_line_3 : REAL;	
	shrpa_voltage_2_line_1 : REAL;	
	shrpa_voltage_2_line_2 : REAL;	
	shrpa_voltage_2_line_3 : REAL;	
	shrpa_voltage_3_line_1 : REAL;	
	shrpa_voltage_4_line_1 : REAL;
	
	shrpa_current_3_line_1 : REAL;	
	shrpa_current_4_line_1 : REAL;
	
	shrpa_freq_3_line_1 : REAL;	
	shrpa_freq_4_line_1 : REAL;
	
	// ЩРПС
	shrps_voltage_registers1: ARRAY [1..6] OF WORD;
	shrps_voltage_registers2: ARRAY [1..6] OF WORD;
	shrps_voltage_registers3: ARRAY [1..6] OF WORD;
	shrps_voltage_registers4: ARRAY [1..6] OF WORD;
	
	Shrps_voltage_1_delay_timer	: TON;
	Shrps_voltage_2_delay_timer	: TON;
	Shrps_voltage_3_delay_timer	: TON;
	Shrps_voltage_4_delay_timer	: TON;
	
	shrps_voltage_1_sum_checker : REAL;
	shrps_voltage_2_sum_checker : REAL;
	shrps_voltage_3_sum_checker : REAL;
	shrps_voltage_4_sum_checker : REAL;

	shrps_voltage_1_line_1 : REAL;
	shrps_voltage_1_line_2 : REAL;
	shrps_voltage_1_line_3 : REAL;
	
	shrps_voltage_2_line_1 : REAL;
	shrps_voltage_2_line_2 : REAL;
	shrps_voltage_2_line_3 : REAL;
	
	shrps_voltage_3_line_1 : REAL;
	shrps_voltage_3_line_2 : REAL;
	shrps_voltage_3_line_3 : REAL;
	
	shrps_voltage_4_line_1 : REAL;
	shrps_voltage_4_line_2 : REAL;
	shrps_voltage_4_line_3 : REAL;


	//Визуализация
	var_true :BOOL := TRUE;
	ack		 :BOOL;
	history  :BOOL;	
	
	//Переменные для работы с климатом
	climate_temp_out          :WORD; 
	climat_temp_out_minus     :BOOL; //Бит отрицательности температуры
	climate_temp_out_real     :REAL; //Наружная температура
	climate_temp_in           :WORD; 
	climat_temp_in_minus      :BOOL; //Бит отрицательности температуры
	climate_temp_in_real      :REAL; //Внутренняя температура
	climate_state_reg         :WORD; 
	climate_state_as_bit      :WORD_AS_BIT;
	climate_zaslonka_state    :BOOL; //Состояние заслонки
	climate_vent_1_state      :BOOL; //Состояние вентилятора №1
	climate_vent_2_state      :BOOL; //Состояние вентилятора №2
	climate_condition_1_state :BOOL; //Состояние кондиционера №1
	climate_condition_2_state :BOOL; //Состояние кондиционера №2
	climate_heat_state        :BOOL; //Состояние обогрева
	climate_heat_door_state   :BOOL; //Состояние обогрева дверей
	climate_auto_state        :BOOL; //Состояние автоматики климата
	climate_temp_excess       :BOOL; //авария. внутренняя температура > 25
	climate_temp_hight		  :BOOL; // 12 бит Высокая температура
	climate_temp_low		  :BOOL; // 11 бит Низкая температура
	
	//Переменные для работы с IPS 1.1
	mpx_a1_power						:WORD := 40;	//Мощность ИБП в кВт
	mpx_a1_time_m						:WORD; //Время автономии в мин
	mpx_a1_1_in_v_1 	 		   		:WORD; //1-е Напряжение входа
	mpx_a1_1_in_v_2 	 		   		:WORD; //2-e Напряжение входа
	mpx_a1_1_in_v_3 	 		   		:WORD; //3-е Напряжение входа
	mpx_a1_1_in_v_1_real 	 		   	:REAL; //1-е Напряжение входа (x0.1)
	mpx_a1_1_in_v_2_real 	 		   	:REAL; //2-e Напряжение входа (x0.1)
	mpx_a1_1_in_v_3_real 	 		   	:REAL; //3-е Напряжение входа (x0.1)
	mpx_a1_1_in_freq 	 		   		:WORD; //Частота на входе
	mpx_a1_1_in_freq_real		   		:REAL; //Частота на входе (x0.1)
	mpx_a1_1_bypass_v_1  		   		:WORD; //1-е Напряжение байпаса
	mpx_a1_1_bypass_v_1_real  		   	:REAL; //1-е Напряжение байпаса (x0.1)
	mpx_a1_1_bypass_freq 		   		:WORD; //Частота байпаса
	mpx_a1_1_bypass_freq_real      		:REAL; //Частота байпаса
	mpx_a1_1_output_v_1  		   		:WORD; //1-е Напряжение выхода
	mpx_a1_1_output_v_1_real  		   	:REAL; //1-е Напряжение выхода (x0.1)
	mpx_a1_1_output_active_power_1 		:word; //Активная мощность 1-й фазы (кВт)
	mpx_a1_1_output_active_power_1_real :REAL; //Активная мощность 1-й фазы (кВт)
	mpx_a1_1_output_freq 	       		:WORD; //Частота выхода
	mpx_a1_1_output_freq_real 	        :REAL; //Частота выхода (x0.1)
	mpx_a1_1_load_ph_1    	       		:WORD; //Загрузска 1-й фазы (%)
	mpx_a1_1_load_ph_1_real    	       	:REAL; //Загрузска 1-й фазы (%) (x0.1)
	mpx_a1_1_battery_voltage 	   		:WORD; //Напряжение батареи
	mpx_a1_1_battery_voltage_real  		:REAL; //Напряжение батареи (x0.1)
	mpx_a1_1_battery_current 	   		:WORD; //Ток батареи
	mpx_a1_1_battery_current_real  		:REAL; //Ток батареи (x0.1)
	mpx_a1_1_battery_capacity 	   		:WORD; //Остаточная емкость батареи (%)
	mpx_a1_1_battery_time 		   		:WORD; //Остаточное время автономии (минуты)
	mpx_a1_1_temp 				   		:WORD; //Температура
	mpx_a1_1_temp_real				   	:REAL; //Температура (x0.1)
	
	mpx_a1_1_Invertor 					:WORD; //Работа от инвертора (14 = ДА, 16 = НЕТ)	
	mpx_a1_1_state_reg 	       			:WORD; //Регистр состояния
	mpx_a1_1_inv_byp					:WORD; //

	mpx_a1_1_bypass_line_state 	   		:STRING; 
	mpx_a1_1_bypass_arrow_state    		:STRING;
	mpx_a1_1_battery_arrow_state 		:STRING; //состояние батареи
	mpx_a1_1_battery_line_state 		:STRING; //состояние батареи
	mpx_a1_1_input_state 		   		:STRING; //состояние входа
	mpx_a1_1_output_state 		   		:STRING; //состояние выхода
	mpx_a1_1_arrow_state 				:STRING;
	mpx_a1_1_alarm                      :BOOL;
	mpx_a1_1_overtemp					:WORD;	
	mpx_a1_1_overload					:WORD;
	mpx_a1_1_outfail					:WORD;
	mpx_a1_1_emergency					:WORD;

	
	//Переменные для работы с IPS 1.2
	mpx_a2_power						:WORD := 40;	//Мощность ИБП в кВт
	mpx_a2_time_m						:WORD; //Время автономии в мин
	mpx_a2_1_in_v_1 	 		   		:WORD; //1-е Напряжение входа
	mpx_a2_1_in_v_2 	 		   		:WORD; //2-e Напряжение входа
	mpx_a2_1_in_v_3 	 		   		:WORD; //3-е Напряжение входа
	mpx_a2_1_in_v_1_real 	 		   	:REAL; //1-е Напряжение входа (x0.1)
	mpx_a2_1_in_v_2_real 	 		   	:REAL; //2-e Напряжение входа (x0.1)
	mpx_a2_1_in_v_3_real 	 		   	:REAL; //3-е Напряжение входа (x0.1)
	mpx_a2_1_in_freq 	 		   		:WORD; //Частота на входе
	mpx_a2_1_in_freq_real		   		:REAL; //Частота на входе (x0.1)
	mpx_a2_1_bypass_v_1  		   		:WORD; //1-е Напряжение байпаса
	mpx_a2_1_bypass_v_1_real  		   	:REAL; //1-е Напряжение байпаса (x0.1)
	mpx_a2_1_bypass_freq 		   		:WORD; //Частота байпаса
	mpx_a2_1_bypass_freq_real      		:REAL; //Частота байпаса
	mpx_a2_1_output_v_1  		   		:WORD; //1-е Напряжение выхода
	mpx_a2_1_output_v_1_real  		   	:REAL; //1-е Напряжение выхода (x0.1)
	mpx_a2_1_output_active_power_1		:WORD;
	mpx_a2_1_output_active_power_1_real :REAL; //Активная мощность 1-й фазы (кВт)
	mpx_a2_1_output_freq 	       		:WORD; //Частота выхода
	mpx_a2_1_output_freq_real 	        :REAL; //Частота выхода (x0.1)
	mpx_a2_1_load_ph_1    	       		:WORD; //Загрузска 1-й фазы (%)
	mpx_a2_1_load_ph_1_real    	       	:REAL; //Загрузска 1-й фазы (%) (x0.1)
	mpx_a2_1_battery_voltage 	   		:WORD; //Напряжение батареи
	mpx_a2_1_battery_voltage_real  		:REAL; //Напряжение батареи (x0.1)
	mpx_a2_1_battery_current 	   		:WORD; //Ток батареи
	mpx_a2_1_battery_current_real  		:REAL; //Ток батареи (x0.1)
	mpx_a2_1_battery_capacity 	   		:WORD; //Остаточная емкость батареи (%)
	mpx_a2_1_battery_time 		   		:WORD; //Остаточное время автономии (минуты)
	mpx_a2_1_temp 				   		:WORD; //Температура
	mpx_a2_1_temp_real				   	:REAL; //Температура (x0.1)
	
	mpx_a2_1_Invertor 					:WORD; //Работа от инвертора (14 = ДА, 16 = НЕТ)	
	mpx_a2_1_state_reg 	       			:WORD; //Регистр состояния
	mpx_a2_1_inv_byp					:WORD; //

	mpx_a2_1_bypass_line_state 	   		:STRING; 
	mpx_a2_1_bypass_arrow_state    		:STRING;
	mpx_a2_1_battery_arrow_state 		:STRING; //состояние батареи
	mpx_a2_1_battery_line_state 		:STRING; //состояние батареи
	mpx_a2_1_input_state 		   		:STRING; //состояние входа
	mpx_a2_1_output_state 		   		:STRING; //состояние выхода
	mpx_a2_1_arrow_state 				:STRING;
	mpx_a2_1_alarm                      :BOOL;
	mpx_a2_1_overtemp					:WORD;	
	mpx_a2_1_overload					:WORD;
	mpx_a2_1_outfail					:WORD;
	mpx_a2_1_emergency					:WORD;
	
	
	//Переменные для работы с IPS 2.1
	mpx_s1_power						:WORD := 150;	//Мощность ИБП в кВт
	mpx_s1_time_m						:WORD; //Время автономии в мин
	mpx_s1_1_in_v_1 	 		   		:WORD; //1-е Напрядение входа
	mpx_s1_1_in_v_2 	 		   		:WORD; //2-e Напряжение входа
	mpx_s1_1_in_v_3 	 		   		:WORD; //3-е Напряжение входа
	mpx_s1_1_in_v_1_real 	 		   	:REAL; //1-е Напрядение входа (x0.1)
	mpx_s1_1_in_v_2_real 	 		   	:REAL; //2-e Напряжение входа (x0.1)
	mpx_s1_1_in_v_3_real 	 		   	:REAL; //3-е Напряжение входа (x0.1)
	mpx_s1_1_in_freq 	 		   		:WORD; //Частота на входе
	mpx_s1_1_in_freq_real		   		:REAL; //Частота на входе (x0.1)
	mpx_s1_1_bypass_v_1  		   		:WORD; //1-е Напряжение байпаса
	mpx_s1_1_bypass_v_2  		   		:WORD; //2-е Напряжение байпаса
	mpx_s1_1_bypass_v_3  		   		:WORD; //3-е Напряжение байпаса
	mpx_s1_1_bypass_v_1_real  		   	:REAL; //1-е Напряжение байпаса (x0.1)
	mpx_s1_1_bypass_v_2_real  		   	:REAL; //2-е Напряжение байпаса (x0.1)
	mpx_s1_1_bypass_v_3_real  		   	:REAL; //3-е Напряжение байпаса (x0.1)
	mpx_s1_1_bypass_freq 		   		:WORD; //Частота байпаса
	mpx_s1_1_bypass_freq_real      		:REAL; //Частота байпаса
	mpx_s1_1_output_v_1  		   		:WORD; //1-е Напряжение выхода
	mpx_s1_1_output_v_2  		   		:WORD; //2-е Напряжение выхода
	mpx_s1_1_output_v_3  		   		:WORD; //3-е Напряжение выхода
	mpx_s1_1_output_v_1_real  		   	:REAL; //1-е Напряжение выхода (x0.1)
	mpx_s1_1_output_v_2_real  		   	:REAL; //2-е Напряжение выхода (x0.1)
	mpx_s1_1_output_v_3_real  		   	:REAL; //3-е Напряжение выхода (x0.1)
	mpx_s1_1_output_active_power_1		:WORD;
	mpx_s1_1_output_active_power_2		:WORD;
	mpx_s1_1_output_active_power_3		:WORD;	
	mpx_s1_1_output_active_power_1_real :REAL; //Активная мощность 1-й фазы (кВт)
	mpx_s1_1_output_active_power_2_real :REAL; //Активная мощность 2-й фазы (кВт)
	mpx_s1_1_output_active_power_3_real :REAL; //Активная мощность 3-й фазы (кВт)
	mpx_s1_1_output_active_power_real   :REAL; //Активная мощность всех фаз
	mpx_s1_1_output_freq 	       		:WORD; //Частота выхода
	mpx_s1_1_output_freq_real 	        :REAL; //Частота выхода (x0.1)
	mpx_s1_1_load_ph_1    	       		:WORD; //Загрузска 1-й фазы (%)
	mpx_s1_1_load_ph_2    		   		:WORD; //Загрузска 3-й фазы (%)
	mpx_s1_1_load_ph_3    	       		:WORD; //Загрузска 2-й фазы (%)
	mpx_s1_1_load_ph_1_real    	       	:REAL; //Загрузска 1-й фазы (%) (x0.1)
	mpx_s1_1_load_ph_2_real    		   	:REAL; //Загрузска 3-й фазы (%) (x0.1)
	mpx_s1_1_load_ph_3_real    	       	:REAL; //Загрузска 2-й фазы (%) (x0.1)
	mpx_s1_1_battery_voltage 	   		:WORD; //Напряжение батареи
	mpx_s1_1_battery_voltage_real  		:REAL; //Напряжение батареи (x0.1)
	mpx_s1_1_battery_current 	   		:WORD; //Ток батареи
	mpx_s1_1_battery_current_real  		:REAL; //Ток батареи (x0.1)
	mpx_s1_1_battery_capacity 	   		:WORD; //Остаточная емкость батареи (%)
	mpx_s1_1_battery_time 		   		:WORD; //Остаточное время автономии (минуты)
	mpx_s1_1_temp 				   		:WORD; //Температура
	mpx_s1_1_temp_real				   	:REAL; //Температура (x0.1)
	
	mpx_s1_1_Invertor 					:WORD; //Работа от инвертора (14 = ДА, 16 = НЕТ)	
	mpx_s1_1_state_reg 	       			:WORD; //Регистр состояния
	mpx_s1_1_inv_byp					:WORD; //

	mpx_s1_1_bypass_line_state 	   		:STRING; 
	mpx_s1_1_bypass_arrow_state    		:STRING;
	mpx_s1_1_battery_arrow_state 		:STRING; //состояние батареи
	mpx_s1_1_battery_line_state 		:STRING; //состояние батареи
	mpx_s1_1_input_state 		   		:STRING; //состояние входа
	mpx_s1_1_output_state 		   		:STRING; //состояние выхода
	mpx_s1_1_arrow_state 				:STRING;
	mpx_s1_1_alarm                      :BOOL;
	mpx_s1_1_overtemp					:WORD;	
	mpx_s1_1_overload					:WORD;
	mpx_s1_1_outfail					:WORD;
	mpx_s1_1_emergency					:WORD;
	
	//Переменные для работы с IPS 2.2
	mpx_s2_power						:WORD := 150;	//Мощность ИБП в кВт
	mpx_s2_time_m						:WORD; //Время автономии в мин
	mpx_s2_1_in_v_1 	 		   		:WORD; //1-е Напрядение входа
	mpx_s2_1_in_v_2 	 		   		:WORD; //2-e Напряжение входа
	mpx_s2_1_in_v_3 	 		   		:WORD; //3-е Напряжение входа
	mpx_s2_1_in_v_1_real 	 		   	:REAL; //1-е Напрядение входа (x0.1)
	mpx_s2_1_in_v_2_real 	 		   	:REAL; //2-e Напряжение входа (x0.1)
	mpx_s2_1_in_v_3_real 	 		   	:REAL; //3-е Напряжение входа (x0.1)
	mpx_s2_1_in_freq 	 		   		:WORD; //Частота на входе
	mpx_s2_1_in_freq_real		   		:REAL; //Частота на входе (x0.1)
	mpx_s2_1_bypass_v_1  		   		:WORD; //1-е Напряжение байпаса
	mpx_s2_1_bypass_v_2  		   		:WORD; //2-е Напряжение байпаса
	mpx_s2_1_bypass_v_3  		   		:WORD; //3-е Напряжение байпаса
	mpx_s2_1_bypass_v_1_real  		   	:REAL; //1-е Напряжение байпаса (x0.1)
	mpx_s2_1_bypass_v_2_real  		   	:REAL; //2-е Напряжение байпаса (x0.1)
	mpx_s2_1_bypass_v_3_real  		   	:REAL; //3-е Напряжение байпаса (x0.1)
	mpx_s2_1_bypass_freq 		   		:WORD; //Частота байпаса
	mpx_s2_1_bypass_freq_real      		:REAL; //Частота байпаса
	mpx_s2_1_output_v_1  		   		:WORD; //1-е Напряжение выхода
	mpx_s2_1_output_v_2  		   		:WORD; //2-е Напряжение выхода
	mpx_s2_1_output_v_3  		   		:WORD; //3-е Напряжение выхода
	mpx_s2_1_output_v_1_real  		   	:REAL; //1-е Напряжение выхода (x0.1)
	mpx_s2_1_output_v_2_real  		   	:REAL; //2-е Напряжение выхода (x0.1)
	mpx_s2_1_output_v_3_real  		   	:REAL; //3-е Напряжение выхода (x0.1)
	mpx_s2_1_output_active_power_1		:WORD;
	mpx_s2_1_output_active_power_2		:WORD;
	mpx_s2_1_output_active_power_3		:WORD;	
	mpx_s2_1_output_active_power_1_real :REAL; //Активная мощность 1-й фазы (кВт)
	mpx_s2_1_output_active_power_2_real :REAL; //Активная мощность 2-й фазы (кВт)
	mpx_s2_1_output_active_power_3_real :REAL; //Активная мощность 3-й фазы (кВт)
	mpx_s2_1_output_active_power_real   :REAL; //Активная мощность всех фаз
	mpx_s2_1_output_freq 	       		:WORD; //Частота выхода
	mpx_s2_1_output_freq_real 	        :REAL; //Частота выхода (x0.1)
	mpx_s2_1_load_ph_1    	       		:WORD; //Загрузска 1-й фазы (%)
	mpx_s2_1_load_ph_2    		   		:WORD; //Загрузска 3-й фазы (%)
	mpx_s2_1_load_ph_3    	       		:WORD; //Загрузска 2-й фазы (%)
	mpx_s2_1_load_ph_1_real    	       	:REAL; //Загрузска 1-й фазы (%) (x0.1)
	mpx_s2_1_load_ph_2_real    		   	:REAL; //Загрузска 3-й фазы (%) (x0.1)
	mpx_s2_1_load_ph_3_real    	       	:REAL; //Загрузска 2-й фазы (%) (x0.1)
	mpx_s2_1_battery_voltage 	   		:WORD; //Напряжение батареи
	mpx_s2_1_battery_voltage_real  		:REAL; //Напряжение батареи (x0.1)
	mpx_s2_1_battery_current 	   		:WORD; //Ток батареи
	mpx_s2_1_battery_current_real  		:REAL; //Ток батареи (x0.1)
	mpx_s2_1_battery_capacity 	   		:WORD; //Остаточная емкость батареи (%)
	mpx_s2_1_battery_time 		   		:WORD; //Остаточное время автономии (минуты)
	mpx_s2_1_temp 				   		:WORD; //Температура
	mpx_s2_1_temp_real				   	:REAL; //Температура (x0.1)
	
	mpx_s2_1_Invertor 					:WORD; //Работа от инвертора (14 = ДА, 16 = НЕТ)	
	mpx_s2_1_state_reg 	       			:WORD; //Регистр состояния
	mpx_s2_1_inv_byp					:WORD; //

	mpx_s2_1_bypass_line_state 	   		:STRING; 
	mpx_s2_1_bypass_arrow_state    		:STRING;
	mpx_s2_1_battery_arrow_state 		:STRING; //состояние батареи
	mpx_s2_1_battery_line_state 		:STRING; //состояние батареи
	mpx_s2_1_input_state 		   		:STRING; //состояние входа
	mpx_s2_1_output_state 		   		:STRING; //состояние выхода
	mpx_s2_1_arrow_state 				:STRING;
	mpx_s2_1_alarm                      :BOOL;
	mpx_s2_1_overtemp					:WORD;	
	mpx_s2_1_overload					:WORD;
	mpx_s2_1_outfail					:WORD;
	mpx_s2_1_emergency					:WORD;			
	
	ips1_1_state						:WORD;
	ips1_2_state						:WORD;
	ips2_1_state						:WORD;
	ips2_2_state						:WORD;
	
	mpx_s1_state_string :WSTRING := "";
	mpx_s2_state_string :WSTRING := "";
	mpx_a1_state_string :WSTRING := "";
	mpx_a2_state_string :WSTRING := "";
	
END_VAR

// Работа с ICP CON
shrps_ups_bus_1 := NOT(shrps_ups_bus_1_raw);
shrps_ups_bus_2 := NOT(shrps_ups_bus_2_raw);
shrpa_ups_in_1 := NOT(shrpa_ups_in_1_raw);
shrpa_ups_in_2 := NOT(shrpa_ups_in_2_raw);

// Работа с ElNet
// ЩРПА
shrpa_voltage_1_sum_checker := shrpa_voltage_registers1[2] + shrpa_voltage_registers1[4] + shrpa_voltage_registers1[6];
Shrpa_voltage_1_delay_timer(IN := (shrpa_voltage_1_sum_checker = 0), PT:= delay_timeout);
IF (Shrpa_voltage_1_delay_timer.Q = TRUE) THEN
	shrpa_voltage_1_line_1 := 0;
	shrpa_voltage_1_line_2 := 0;
	shrpa_voltage_1_line_3 := 0;
ELSIF (shrpa_voltage_1_sum_checker > 0) THEN
	shrpa_voltage_1_line_1 := shrpa_voltage_registers1[2];
	shrpa_voltage_1_line_2 := shrpa_voltage_registers1[4];
	shrpa_voltage_1_line_3 := shrpa_voltage_registers1[6];
END_IF

shrpa_voltage_2_sum_checker := shrpa_voltage_registers2[2] + shrpa_voltage_registers2[4] + shrpa_voltage_registers2[6];
Shrpa_voltage_2_delay_timer(IN := (shrpa_voltage_2_sum_checker = 0), PT:= delay_timeout);
IF (Shrpa_voltage_2_delay_timer.Q = TRUE) THEN
	shrpa_voltage_2_line_1 := 0;
	shrpa_voltage_2_line_2 := 0;
	shrpa_voltage_2_line_3 := 0;
ELSIF (shrpa_voltage_2_sum_checker > 0) THEN
	shrpa_voltage_2_line_1 := shrpa_voltage_registers2[2];
	shrpa_voltage_2_line_2 := shrpa_voltage_registers2[4];
	shrpa_voltage_2_line_3 := shrpa_voltage_registers2[6];
END_IF

Shrpa_voltage_3_delay_timer(IN := (shrpa_voltage_registers3[2] = 0), PT:= delay_timeout);
IF (Shrpa_voltage_3_delay_timer.Q = TRUE) THEN
	shrpa_voltage_3_line_1 := 0;
	shrpa_current_3_line_1 := 0;
	shrpa_freq_3_line_1 := 0;
ELSIF (shrpa_voltage_registers3[2] > 0) THEN
	shrpa_voltage_3_line_1 := shrpa_voltage_registers3[2];
	shrpa_current_3_line_1 := shrpa_current_registers3[2];
	shrpa_freq_3_line_1 := shrpa_freq_registers3[2];
END_IF

Shrpa_voltage_4_delay_timer(IN := (shrpa_voltage_registers4[2] = 0), PT:= delay_timeout);
IF (Shrpa_voltage_4_delay_timer.Q = TRUE) THEN
	shrpa_voltage_4_line_1 := 0;
	shrpa_current_4_line_1 := 0;
	shrpa_freq_4_line_1 := 0;
ELSIF (shrpa_voltage_registers4[2] > 0) THEN
	shrpa_voltage_4_line_1 := shrpa_voltage_registers4[2];
	shrpa_current_4_line_1 := shrpa_current_registers4[2];
	shrpa_freq_4_line_1 := shrpa_freq_registers4[2];
END_IF

// ЩРПС
shrps_voltage_1_sum_checker := shrps_voltage_registers1[2] + shrps_voltage_registers1[4] + shrps_voltage_registers1[6];
Shrps_voltage_1_delay_timer(IN := (shrps_voltage_1_sum_checker = 0), PT:= delay_timeout);
IF (Shrps_voltage_1_delay_timer.Q = TRUE) THEN
	shrps_voltage_1_line_1 := 0;
	shrps_voltage_1_line_2 := 0;
	shrps_voltage_1_line_3 := 0;
ELSIF (shrps_voltage_1_sum_checker > 0) THEN
	shrps_voltage_1_line_1 := shrps_voltage_registers1[2];
	shrps_voltage_1_line_2 := shrps_voltage_registers1[4];
	shrps_voltage_1_line_3 := shrps_voltage_registers1[6];
END_IF

shrps_voltage_2_sum_checker := shrps_voltage_registers2[2] + shrps_voltage_registers2[4] + shrps_voltage_registers2[6];
Shrps_voltage_2_delay_timer(IN := (shrps_voltage_2_sum_checker = 0), PT:= delay_timeout);
IF (Shrps_voltage_2_delay_timer.Q = TRUE) THEN
	shrps_voltage_2_line_1 := 0;
	shrps_voltage_2_line_2 := 0;
	shrps_voltage_2_line_3 := 0;
ELSIF (shrps_voltage_2_sum_checker > 0) THEN
	shrps_voltage_2_line_1 := shrps_voltage_registers2[2];
	shrps_voltage_2_line_2 := shrps_voltage_registers2[4];
	shrps_voltage_2_line_3 := shrps_voltage_registers2[6];
END_IF

shrps_voltage_3_sum_checker := shrps_voltage_registers3[2] + shrps_voltage_registers3[4] + shrps_voltage_registers3[6];
Shrps_voltage_3_delay_timer(IN := (shrps_voltage_3_sum_checker = 0), PT:= delay_timeout);
IF (Shrps_voltage_3_delay_timer.Q = TRUE) THEN
	shrps_voltage_3_line_1 := 0;
	shrps_voltage_3_line_2 := 0;
	shrps_voltage_3_line_3 := 0;
ELSIF (shrps_voltage_3_sum_checker > 0) THEN
	shrps_voltage_3_line_1 := shrps_voltage_registers3[2];
	shrps_voltage_3_line_2 := shrps_voltage_registers3[4];
	shrps_voltage_3_line_3 := shrps_voltage_registers3[6];
END_IF

shrps_voltage_4_sum_checker := shrps_voltage_registers4[2] + shrps_voltage_registers4[4] + shrps_voltage_registers4[6];
Shrps_voltage_4_delay_timer(IN := (shrps_voltage_4_sum_checker = 0), PT:= delay_timeout);
IF (Shrps_voltage_4_delay_timer.Q = TRUE) THEN
	shrps_voltage_4_line_1 := 0;
	shrps_voltage_4_line_2 := 0;
	shrps_voltage_4_line_3 := 0;
ELSIF (shrps_voltage_4_sum_checker > 0) THEN
	shrps_voltage_4_line_1 := shrps_voltage_registers4[2];
	shrps_voltage_4_line_2 := shrps_voltage_registers4[4];
	shrps_voltage_4_line_3 := shrps_voltage_registers4[6];
END_IF

//Работа с климатом
climate_state_as_bit(W    := climate_state_reg);
climate_zaslonka_state    := climate_state_as_bit.B03;
climate_vent_1_state      := climate_state_as_bit.B00;
climate_vent_2_state      := climate_state_as_bit.B01;
climate_condition_1_state := climate_state_as_bit.B04;
climate_condition_2_state := climate_state_as_bit.B05;
climate_heat_state        := climate_state_as_bit.B02;
climate_heat_door_state   := climate_state_as_bit.B06;
climate_auto_state        := NOT(climate_state_as_bit.B07);
climat_temp_out_minus     := climate_state_as_bit.B10;
climat_temp_in_minus      := climate_state_as_bit.B09;
climate_temp_low      	  := climate_state_as_bit.B11;
climate_temp_hight        := climate_state_as_bit.B12;

climate_temp_out_real     := climate_temp_out * 0.1;
climate_temp_in_real      := climate_temp_in * 0.1;
IF (climat_temp_out_minus = TRUE) THEN
	climate_temp_out_real := climate_temp_out_real * (-1);
END_IF
IF (climat_temp_in_minus = TRUE) THEN
	climate_temp_in_real := climate_temp_in_real * (-1);
END_IF
IF (climate_temp_in_real > 25) THEN
	climate_temp_excess := TRUE;
	ELSE
		climate_temp_excess := FALSE;
END_IF

//------------------------------------IPS 1.1-------------------------------------
//Конвертация параметров IPS 1.1
mpx_a1_1_in_v_1_real 	 		   	:= mpx_a1_1_in_v_1 * 0.1;
mpx_a1_1_in_v_2_real 	 			:= mpx_a1_1_in_v_2 * 0.1;   		
mpx_a1_1_in_v_3_real 	 		 	:= mpx_a1_1_in_v_3 * 0.1;  		
mpx_a1_1_in_freq_real               := mpx_a1_1_in_freq * 0.1;

mpx_a1_1_bypass_v_1_real			:= mpx_a1_1_bypass_v_1 * 0.1;
mpx_a1_1_bypass_freq_real           := mpx_a1_1_bypass_freq * 0.1;

mpx_a1_1_output_v_1_real			:= mpx_a1_1_output_v_1 * 0.1;
mpx_a1_1_output_freq_real           := mpx_a1_1_output_freq * 0.1;

mpx_a1_1_load_ph_1_real				:= mpx_a1_1_load_ph_1 * 0.1;
mpx_a1_1_output_active_power_1_real	:= mpx_a1_power * mpx_a1_1_load_ph_1_real * 0.01;

mpx_a1_1_output_active_power_1 		:= REAL_TO_WORD(mpx_a1_1_output_active_power_1_real * 1000);

mpx_a1_1_battery_voltage_real       := mpx_a1_1_battery_voltage * 1;
mpx_a1_1_battery_current_real       := mpx_a1_1_battery_current * 0.1;

mpx_a1_1_temp_real 					:= mpx_a1_1_temp * 0.1;


//Логика состояний IPS 1.1
IF ((mpx_a1_1_Invertor = 14) AND (mpx_a1_1_state_reg = 2) AND (mpx_a1_1_inv_byp = 12)) THEN
	mpx_a1_1_bypass_line_state := 'bypass_line1_off';
	mpx_a1_1_bypass_arrow_state := 'bypass_arrow_off';
	mpx_a1_1_input_state := 'arrow_on';	
	mpx_a1_1_output_state := 'arrow_on';
	mpx_a1_1_arrow_state := 'arrow_on';
	mpx_a1_1_battery_line_state := 'battery_line_on';
	mpx_a1_1_battery_arrow_state := 'battery_arrow_on';
	mpx_a1_state_string := "От сети";	
	ips1_1_state := 1;
ELSE
	IF ((mpx_a1_1_Invertor = 14) AND (mpx_a1_1_state_reg = 3) AND (mpx_a1_1_inv_byp = 12)) THEN	
		mpx_a1_1_bypass_line_state := 'bypass_line1_off';
		mpx_a1_1_bypass_arrow_state := 'bypass_arrow_off';
		mpx_a1_1_input_state := 'arrow_off';
		mpx_a1_1_output_state := 'arrow_on';
		mpx_a1_1_arrow_state := 'arrow_on';
		mpx_a1_1_battery_line_state := 'battery_line_on';
		mpx_a1_1_battery_arrow_state := 'battery_arrow_on';
		mpx_a1_state_string := "От АКБ";
		ips1_1_state := 2;	
	ELSE	
		IF ((mpx_a1_1_Invertor = 16) AND (mpx_a1_1_state_reg = 3) AND (mpx_a1_1_inv_byp = 13)) THEN	
			mpx_a1_1_bypass_line_state := 'bypass_line_on';
			mpx_a1_1_bypass_arrow_state := 'bypass_arrow_on';
			mpx_a1_1_input_state := 'arrow_off';
			mpx_a1_1_output_state := 'arrow_on';
			mpx_a1_1_arrow_state := 'arrow_off';
			mpx_a1_1_battery_line_state := 'battery_line_off';
			mpx_a1_1_battery_arrow_state := 'battery_arrow_off';
			mpx_a1_state_string := "Байпас";
			ips1_1_state := 3;	
		ELSE	
			IF ((mpx_a1_1_Invertor = 14) AND (mpx_a1_1_state_reg = 2) AND (mpx_a1_1_inv_byp = 13)) THEN	
				mpx_a1_1_bypass_line_state := 'bypass_line_on';
				mpx_a1_1_bypass_arrow_state := 'bypass_arrow_on';
				mpx_a1_1_input_state := 'arrow_off';
				mpx_a1_1_output_state := 'arrow_on';
				mpx_a1_1_arrow_state := 'arrow_off';
				mpx_a1_1_battery_line_state := 'battery_line_off';
				mpx_a1_1_battery_arrow_state := 'battery_arrow_off';
				mpx_a1_state_string := "Байпас";
				ips1_1_state := 3;	
			ELSE	
				mpx_a1_1_bypass_line_state := 'bypass_line1_off';
				mpx_a1_1_bypass_arrow_state := 'bypass_arrow_off';
				mpx_a1_1_input_state := 'arrow_off';
				mpx_a1_1_output_state := 'arrow_off';
				mpx_a1_1_arrow_state := 'arrow_off';
				mpx_a1_1_battery_line_state := 'battery_line_off';
				mpx_a1_1_battery_arrow_state := 'battery_arrow_off';
				mpx_a1_state_string := "Неизвестно";
				ips1_1_state := 0;
			END_IF
		END_IF
	END_IF
END_IF

IF ((mpx_a1_1_overtemp = 14) OR (mpx_a1_1_overload = 14) OR (mpx_a1_1_outfail = 14) OR (mpx_a1_1_emergency = 14)) THEN
	mpx_a1_1_alarm := TRUE;
ELSE
	mpx_a1_1_alarm := FALSE;
END_IF

//------------------------------------IPS 1.2-------------------------------------
//Конвертация параметров IPS 1.2
mpx_a2_1_in_v_1_real 	 		   	:= mpx_a2_1_in_v_1 * 0.1;
mpx_a2_1_in_v_2_real 	 			:= mpx_a2_1_in_v_2 * 0.1;   		
mpx_a2_1_in_v_3_real 	 		 	:= mpx_a2_1_in_v_3 * 0.1;  		
mpx_a2_1_in_freq_real               := mpx_a2_1_in_freq * 0.1;

mpx_a2_1_bypass_v_1_real			:= mpx_a2_1_bypass_v_1 * 0.1;
mpx_a2_1_bypass_freq_real           := mpx_a2_1_bypass_freq * 0.1;

mpx_a2_1_output_v_1_real			:= mpx_a2_1_output_v_1 * 0.1;
mpx_a2_1_output_freq_real           := mpx_a2_1_output_freq * 0.1;

mpx_a2_1_load_ph_1_real				:= mpx_a2_1_load_ph_1 * 0.1;
mpx_a2_1_output_active_power_1_real	:= mpx_a2_power * mpx_a2_1_load_ph_1_real * 0.01;

mpx_a2_1_output_active_power_1 		:= REAL_TO_WORD(mpx_a2_1_output_active_power_1_real * 1000);

mpx_a2_1_battery_voltage_real       := mpx_a2_1_battery_voltage * 1;
mpx_a2_1_battery_current_real       := mpx_a2_1_battery_current * 0.1;

mpx_a2_1_temp_real 					:= mpx_a2_1_temp * 0.1;


//Логика состояний IPS 1.2
IF ((mpx_a2_1_Invertor = 14) AND (mpx_a2_1_state_reg = 2) AND (mpx_a2_1_inv_byp = 12)) THEN
	mpx_a2_1_bypass_line_state := 'bypass_line1_off';
	mpx_a2_1_bypass_arrow_state := 'bypass_arrow_off';
	mpx_a2_1_input_state := 'arrow_on';	
	mpx_a2_1_output_state := 'arrow_on';
	mpx_a2_1_arrow_state := 'arrow_on';
	mpx_a2_1_battery_line_state := 'battery_line_on';
	mpx_a2_1_battery_arrow_state := 'battery_arrow_on';
	mpx_a2_state_string := "От сети";	
	ips1_2_state := 1;
ELSE
	IF ((mpx_a2_1_Invertor = 14) AND (mpx_a2_1_state_reg = 3) AND (mpx_a2_1_inv_byp = 12)) THEN	
		mpx_a2_1_bypass_line_state := 'bypass_line1_off';
		mpx_a2_1_bypass_arrow_state := 'bypass_arrow_off';
		mpx_a2_1_input_state := 'arrow_off';
		mpx_a2_1_output_state := 'arrow_on';
		mpx_a2_1_arrow_state := 'arrow_on';
		mpx_a2_1_battery_line_state := 'battery_line_on';
		mpx_a2_1_battery_arrow_state := 'battery_arrow_on';
		mpx_a2_state_string := "От АКБ";
		ips1_2_state := 2;	
	ELSE	
		IF ((mpx_a2_1_Invertor = 16) AND (mpx_a2_1_state_reg = 3) AND (mpx_a2_1_inv_byp = 13)) THEN	
			mpx_a2_1_bypass_line_state := 'bypass_line_on';
			mpx_a2_1_bypass_arrow_state := 'bypass_arrow_on';
			mpx_a2_1_input_state := 'arrow_off';
			mpx_a2_1_output_state := 'arrow_on';
			mpx_a2_1_arrow_state := 'arrow_off';
			mpx_a2_1_battery_line_state := 'battery_line_off';
			mpx_a2_1_battery_arrow_state := 'battery_arrow_off';
			mpx_a2_state_string := "Байпас";
			ips1_2_state := 3;	
		ELSE	
			IF ((mpx_a2_1_Invertor = 14) AND (mpx_a2_1_state_reg = 2) AND (mpx_a2_1_inv_byp = 13)) THEN	
				mpx_a2_1_bypass_line_state := 'bypass_line_on';
				mpx_a2_1_bypass_arrow_state := 'bypass_arrow_on';
				mpx_a2_1_input_state := 'arrow_off';
				mpx_a2_1_output_state := 'arrow_on';
				mpx_a2_1_arrow_state := 'arrow_off';
				mpx_a2_1_battery_line_state := 'battery_line_off';
				mpx_a2_1_battery_arrow_state := 'battery_arrow_off';
				mpx_a2_state_string := "Байпас";
				ips1_2_state := 3;	
			ELSE	
				mpx_a2_1_bypass_line_state := 'bypass_line1_off';
				mpx_a2_1_bypass_arrow_state := 'bypass_arrow_off';
				mpx_a2_1_input_state := 'arrow_off';
				mpx_a2_1_output_state := 'arrow_off';
				mpx_a2_1_arrow_state := 'arrow_off';
				mpx_a2_1_battery_line_state := 'battery_line_off';
				mpx_a2_1_battery_arrow_state := 'battery_arrow_off';
				mpx_a2_state_string := "Неизвестно";
				ips1_2_state := 0;
			END_IF
		END_IF
	END_IF
END_IF



IF ((mpx_a2_1_overtemp = 14) OR (mpx_a2_1_overload = 14) OR (mpx_a2_1_outfail = 14) OR (mpx_a2_1_emergency = 14)) THEN
	mpx_a2_1_alarm := TRUE;
ELSE
	mpx_a2_1_alarm := FALSE;
END_IF


//------------------------------------IPS 2.1-------------------------------------
//Конвертация параметров IPS 2.1
mpx_s1_1_in_v_1_real 	 		   	:= mpx_s1_1_in_v_1 * 0.1;
mpx_s1_1_in_v_2_real 	 			:= mpx_s1_1_in_v_2 * 0.1;   		
mpx_s1_1_in_v_3_real 	 		 	:= mpx_s1_1_in_v_3 * 0.1;  		
mpx_s1_1_in_freq_real               := mpx_s1_1_in_freq * 0.1;

mpx_s1_1_bypass_v_1_real			:= mpx_s1_1_bypass_v_1 * 0.1;
mpx_s1_1_bypass_v_2_real			:= mpx_s1_1_bypass_v_2 * 0.1;
mpx_s1_1_bypass_v_3_real			:= mpx_s1_1_bypass_v_3 * 0.1;
mpx_s1_1_bypass_freq_real           := mpx_s1_1_bypass_freq * 0.1;

mpx_s1_1_output_v_1_real			:= mpx_s1_1_output_v_1 * 0.1;
mpx_s1_1_output_v_2_real			:= mpx_s1_1_output_v_2 * 0.1;
mpx_s1_1_output_v_3_real			:= mpx_s1_1_output_v_3 * 0.1;
mpx_s1_1_output_freq_real           := mpx_s1_1_output_freq * 0.1;

mpx_s1_1_load_ph_1_real				:= mpx_s1_1_load_ph_1 * 0.1;
mpx_s1_1_load_ph_2_real				:= mpx_s1_1_load_ph_2 * 0.1;
mpx_s1_1_load_ph_3_real				:= mpx_s1_1_load_ph_3 * 0.1;

mpx_s1_1_output_active_power_1_real	:= mpx_s1_power * mpx_s1_1_load_ph_1_real * 0.01;
mpx_s1_1_output_active_power_2_real	:= mpx_s1_power * mpx_s1_1_load_ph_2_real * 0.01;
mpx_s1_1_output_active_power_3_real	:= mpx_s1_power * mpx_s1_1_load_ph_3_real * 0.01;

mpx_s1_1_output_active_power_1 		:= REAL_TO_WORD(mpx_s1_1_output_active_power_1_real * 1000);
mpx_s1_1_output_active_power_2 		:= REAL_TO_WORD(mpx_s1_1_output_active_power_2_real * 1000);
mpx_s1_1_output_active_power_3 		:= REAL_TO_WORD(mpx_s1_1_output_active_power_3_real * 1000);

mpx_s1_1_battery_voltage_real       := mpx_s1_1_battery_voltage * 1;
mpx_s1_1_battery_current_real       := mpx_s1_1_battery_current * 0.1;

mpx_s1_1_temp_real 					:= mpx_s1_1_temp * 0.1;

//Логика состояний IPS 2.1
IF ((mpx_s1_1_Invertor = 14) AND (mpx_s1_1_state_reg = 2) AND (mpx_s1_1_inv_byp = 12)) THEN
	mpx_s1_1_bypass_line_state := 'bypass_line1_off';
	mpx_s1_1_bypass_arrow_state := 'bypass_arrow_off';
	mpx_s1_1_input_state := 'arrow_on';	
	mpx_s1_1_output_state := 'arrow_on';
	mpx_s1_1_arrow_state := 'arrow_on';
	mpx_s1_1_battery_line_state := 'battery_line_on';
	mpx_s1_1_battery_arrow_state := 'battery_arrow_on';
	mpx_s1_state_string := "От сети";	
	ips2_1_state := 1;
ELSE
	IF ((mpx_s1_1_Invertor = 14) AND (mpx_s1_1_state_reg = 3) AND (mpx_s1_1_inv_byp = 12)) THEN	
		mpx_s1_1_bypass_line_state := 'bypass_line1_off';
		mpx_s1_1_bypass_arrow_state := 'bypass_arrow_off';
		mpx_s1_1_input_state := 'arrow_off';
		mpx_s1_1_output_state := 'arrow_on';
		mpx_s1_1_arrow_state := 'arrow_on';
		mpx_s1_1_battery_line_state := 'battery_line_on';
		mpx_s1_1_battery_arrow_state := 'battery_arrow_on';
		mpx_s1_state_string := "От АКБ";
		ips2_1_state := 2;	
	ELSE	
		IF ((mpx_s1_1_Invertor = 16) AND (mpx_s1_1_state_reg = 3) AND (mpx_s1_1_inv_byp = 13)) THEN	
			mpx_s1_1_bypass_line_state := 'bypass_line_on';
			mpx_s1_1_bypass_arrow_state := 'bypass_arrow_on';
			mpx_s1_1_input_state := 'arrow_off';
			mpx_s1_1_output_state := 'arrow_on';
			mpx_s1_1_arrow_state := 'arrow_off';
			mpx_s1_1_battery_line_state := 'battery_line_off';
			mpx_s1_1_battery_arrow_state := 'battery_arrow_off';
			mpx_s1_state_string := "Байпас";
			ips2_1_state := 3;	
		ELSE	
			IF ((mpx_s1_1_Invertor = 14) AND (mpx_s1_1_state_reg = 2) AND (mpx_s1_1_inv_byp = 13)) THEN	
				mpx_s1_1_bypass_line_state := 'bypass_line_on';
				mpx_s1_1_bypass_arrow_state := 'bypass_arrow_on';
				mpx_s1_1_input_state := 'arrow_off';
				mpx_s1_1_output_state := 'arrow_on';
				mpx_s1_1_arrow_state := 'arrow_off';
				mpx_s1_1_battery_line_state := 'battery_line_off';
				mpx_s1_1_battery_arrow_state := 'battery_arrow_off';
				mpx_s1_state_string := "Байпас";
				ips2_1_state := 3;	
			ELSE	
				mpx_s1_1_bypass_line_state := 'bypass_line1_off';
				mpx_s1_1_bypass_arrow_state := 'bypass_arrow_off';
				mpx_s1_1_input_state := 'arrow_off';
				mpx_s1_1_output_state := 'arrow_off';
				mpx_s1_1_arrow_state := 'arrow_off';
				mpx_s1_1_battery_line_state := 'battery_line_off';
				mpx_s1_1_battery_arrow_state := 'battery_arrow_off';
				mpx_s1_state_string := "Неизвестно";
				ips2_1_state := 0;
			END_IF
		END_IF
	END_IF
END_IF


IF ((mpx_s1_1_overtemp = 14) OR (mpx_s1_1_overload = 14) OR (mpx_s1_1_outfail = 14) OR (mpx_s1_1_emergency = 14)) THEN
	mpx_s1_1_alarm := TRUE;
ELSE
	mpx_s1_1_alarm := FALSE;
END_IF

//------------------------------------IPS 2.2-------------------------------------
//Конвертация параметров IPS 2.2
mpx_s2_1_in_v_1_real 	 		   	:= mpx_s2_1_in_v_1 * 0.1;
mpx_s2_1_in_v_2_real 	 			:= mpx_s2_1_in_v_2 * 0.1;   		
mpx_s2_1_in_v_3_real 	 		 	:= mpx_s2_1_in_v_3 * 0.1;  		
mpx_s2_1_in_freq_real               := mpx_s2_1_in_freq * 0.1;

mpx_s2_1_bypass_v_1_real			:= mpx_s2_1_bypass_v_1 * 0.1;
mpx_s2_1_bypass_v_2_real			:= mpx_s2_1_bypass_v_2 * 0.1;
mpx_s2_1_bypass_v_3_real			:= mpx_s2_1_bypass_v_3 * 0.1;
mpx_s2_1_bypass_freq_real           := mpx_s2_1_bypass_freq * 0.1;

mpx_s2_1_output_v_1_real			:= mpx_s2_1_output_v_1 * 0.1;
mpx_s2_1_output_v_2_real			:= mpx_s2_1_output_v_2 * 0.1;
mpx_s2_1_output_v_3_real			:= mpx_s2_1_output_v_3 * 0.1;
mpx_s2_1_output_freq_real           := mpx_s2_1_output_freq * 0.1;

mpx_s2_1_load_ph_1_real				:= mpx_s2_1_load_ph_1 * 0.1;
mpx_s2_1_load_ph_2_real				:= mpx_s2_1_load_ph_2 * 0.1;
mpx_s2_1_load_ph_3_real				:= mpx_s2_1_load_ph_3 * 0.1;

mpx_s2_1_output_active_power_1_real	:= mpx_s2_power * mpx_s2_1_load_ph_1_real * 0.01;
mpx_s2_1_output_active_power_2_real	:= mpx_s2_power * mpx_s2_1_load_ph_2_real * 0.01;
mpx_s2_1_output_active_power_3_real	:= mpx_s2_power * mpx_s2_1_load_ph_3_real * 0.01;

mpx_s2_1_output_active_power_1 		:= REAL_TO_WORD(mpx_s2_1_output_active_power_1_real * 1000);
mpx_s2_1_output_active_power_2 		:= REAL_TO_WORD(mpx_s2_1_output_active_power_2_real * 1000);
mpx_s2_1_output_active_power_3 		:= REAL_TO_WORD(mpx_s2_1_output_active_power_3_real * 1000);

mpx_s2_1_output_active_power_real := mpx_s2_1_output_active_power_1_real + mpx_s2_1_output_active_power_2_real + mpx_s2_1_output_active_power_3_real;

mpx_s2_1_battery_voltage_real       := mpx_s2_1_battery_voltage * 1;
mpx_s2_1_battery_current_real       := mpx_s2_1_battery_current * 0.1;

mpx_s2_1_temp_real 					:= mpx_s2_1_temp * 0.1;

//Логика состояний MPX_s2_1
IF ((mpx_s2_1_Invertor = 14) AND (mpx_s2_1_state_reg = 2) AND (mpx_s2_1_inv_byp = 12)) THEN
	mpx_s2_1_bypass_line_state := 'bypass_line1_off';
	mpx_s2_1_bypass_arrow_state := 'bypass_arrow_off';
	mpx_s2_1_input_state := 'arrow_on';	
	mpx_s2_1_output_state := 'arrow_on';
	mpx_s2_1_arrow_state := 'arrow_on';
	mpx_s2_1_battery_line_state := 'battery_line_on';
	mpx_s2_1_battery_arrow_state := 'battery_arrow_on';
	mpx_s2_state_string := "От сети";	
	ips2_2_state := 1;
ELSE
	IF ((mpx_s2_1_Invertor = 14) AND (mpx_s2_1_state_reg = 3) AND (mpx_s2_1_inv_byp = 12)) THEN	
		mpx_s2_1_bypass_line_state := 'bypass_line1_off';
		mpx_s2_1_bypass_arrow_state := 'bypass_arrow_off';
		mpx_s2_1_input_state := 'arrow_off';
		mpx_s2_1_output_state := 'arrow_on';
		mpx_s2_1_arrow_state := 'arrow_on';
		mpx_s2_1_battery_line_state := 'battery_line_on';
		mpx_s2_1_battery_arrow_state := 'battery_arrow_on';
		mpx_s2_state_string := "От АКБ";
		ips2_2_state := 2;	
	ELSE	
		IF ((mpx_s2_1_Invertor = 16) AND (mpx_s2_1_state_reg = 3) AND (mpx_s2_1_inv_byp = 13)) THEN	
			mpx_s2_1_bypass_line_state := 'bypass_line_on';
			mpx_s2_1_bypass_arrow_state := 'bypass_arrow_on';
			mpx_s2_1_input_state := 'arrow_off';
			mpx_s2_1_output_state := 'arrow_on';
			mpx_s2_1_arrow_state := 'arrow_off';
			mpx_s2_1_battery_line_state := 'battery_line_off';
			mpx_s2_1_battery_arrow_state := 'battery_arrow_off';
			mpx_s2_state_string := "Байпас";
			ips2_2_state := 3;	
		ELSE	
			IF ((mpx_s2_1_Invertor = 14) AND (mpx_s2_1_state_reg = 2) AND (mpx_s2_1_inv_byp = 13)) THEN	
				mpx_s2_1_bypass_line_state := 'bypass_line_on';
				mpx_s2_1_bypass_arrow_state := 'bypass_arrow_on';
				mpx_s2_1_input_state := 'arrow_off';
				mpx_s2_1_output_state := 'arrow_on';
				mpx_s2_1_arrow_state := 'arrow_off';
				mpx_s2_1_battery_line_state := 'battery_line_off';
				mpx_s2_1_battery_arrow_state := 'battery_arrow_off';
				mpx_s2_state_string := "Байпас";
				ips2_2_state := 3;	
			ELSE	
				mpx_s2_1_bypass_line_state := 'bypass_line1_off';
				mpx_s2_1_bypass_arrow_state := 'bypass_arrow_off';
				mpx_s2_1_input_state := 'arrow_off';
				mpx_s2_1_output_state := 'arrow_off';
				mpx_s2_1_arrow_state := 'arrow_off';
				mpx_s2_1_battery_line_state := 'battery_line_off';
				mpx_s2_1_battery_arrow_state := 'battery_arrow_off';
				mpx_s2_state_string := "Неизвестно";
				ips2_2_state := 0;
			END_IF
		END_IF
	END_IF
END_IF



IF ((mpx_s2_1_overtemp = 14) OR (mpx_s2_1_overload = 14) OR (mpx_s2_1_outfail = 14) OR (mpx_s2_1_emergency = 14)) THEN
	mpx_s2_1_alarm := TRUE;
ELSE
	mpx_s2_1_alarm := FALSE;
END_IF

END_PROGRAM

// CODESYS_Control_for_Raspberry_Pi/Application/GPIO_HANDLER
PROGRAM GPIO_HANDLER
VAR
	
	IN_1: BOOL; // ШОПС: Нарушение ШОС	
	IN_2: BOOL; // ШОПС: Пожар
	IN_3: BOOL; // ШОПС: Неисправность ШОС	
	IN_4: BOOL; // ШАСН: Наличие напряжения на 1 вводе	
	IN_5: BOOL; // ШАСН: Наличие напряжения на 2 вводе	
	IN_6: BOOL; // ШАСН: Наличие напряжения на шине БП
	IN_7: BOOL; // ШАСН: Наличие напряжения на шине ГП
	IN_8: BOOL; // ШАСН: Обогрев в УГП включен	
	IN_9: BOOL; // ШАСН: QS1 в первом положении	
	IN_10: BOOL; // ШАСН: QS1 во втором положении
	IN_11: BOOL; // ШАСН: QFV1 включен
	IN_12: BOOL;  // ШАСН: QFV2 включен
	
	RAW_IN_1: BOOL;
	RAW_IN_2: BOOL;
	RAW_IN_3: BOOL; 
	RAW_IN_4: BOOL; 
	RAW_IN_5: BOOL; 
	RAW_IN_6: BOOL; 
	RAW_IN_7: BOOL; 
	RAW_IN_8: BOOL;
	RAW_IN_9: BOOL;
	RAW_IN_10: BOOL;
	RAW_IN_11: BOOL;
	RAW_IN_12: BOOL; 
END_VAR

 IN_1 := NOT(RAW_IN_1);
 IN_2 := NOT(RAW_IN_2);
 IN_3 := NOT(RAW_IN_3);
 IN_4 := NOT(RAW_IN_4);
 IN_5 := NOT(RAW_IN_5);
 IN_6 := NOT(RAW_IN_6);
 IN_7 := NOT(RAW_IN_7);
 IN_8 := NOT(RAW_IN_8);
 IN_9 := NOT(RAW_IN_9);
 IN_10 := NOT(RAW_IN_10);
 IN_11 := NOT(RAW_IN_11);
 IN_12 := NOT(RAW_IN_12);

END_PROGRAM

// CODESYS_Control_for_Raspberry_Pi/Application/AlarmChecker
PROGRAM AlarmChecker
VAR
	MIN_VOLTAGE : WORD := 50;
	
	ups_s1_in_v_alarm : BOOL;
	ups_s2_in_v_alarm : BOOL;
	ups_a1_in_v_alarm : BOOL;
	ups_a2_in_v_alarm : BOOL;
	
	ups_s1_out_v_alarm : BOOL;
	ups_s2_out_v_alarm : BOOL;
	ups_a1_out_v_alarm : BOOL;
	ups_a2_out_v_alarm : BOOL;
	
	shasn_alarm        : BOOL;
	schrpa_alarm       : BOOL;
	schrps_alarm       : BOOL;
	
	schrps_alarm_raw       	: BOOL;
	Shrps_delay_timer		: TON;

	delay_timeout 			: TIME := T#5S;
	
	shrpa_in_1_alarm	: BOOL;
	shrpa_in_2_alarm	: BOOL;
	shrpa_out_alarm		: BOOL;
	
	shrps_in_1_alarm	: BOOL;
	shrps_in_2_alarm	: BOOL;
	shrps_out_alarm		: BOOL;
	shrps_out_alarm_raw	: BOOL;
END_VAR

//Авария входного напряжения ИБПС1
IF( (PLC_PRG.mpx_s1_1_in_v_1 < MIN_VOLTAGE) OR (PLC_PRG.mpx_s1_1_in_v_2 < MIN_VOLTAGE) OR (PLC_PRG.mpx_s1_1_in_v_3 < MIN_VOLTAGE)) THEN
	ups_s1_in_v_alarm := TRUE;
ELSE
	ups_s1_in_v_alarm := FALSE;
END_IF

//Авария входного напряжения ИБПС2
IF((PLC_PRG.mpx_s2_1_in_v_1 < MIN_VOLTAGE) OR (PLC_PRG.mpx_s2_1_in_v_2 < MIN_VOLTAGE) OR (PLC_PRG.mpx_s2_1_in_v_3 < MIN_VOLTAGE)) THEN
	ups_s2_in_v_alarm := TRUE;
ELSE
	ups_s2_in_v_alarm := FALSE;
END_IF

//Авария входного напряжения ИБПА1
IF( (PLC_PRG.mpx_a1_1_in_v_1 < MIN_VOLTAGE) OR (PLC_PRG.mpx_a1_1_in_v_2 < MIN_VOLTAGE) OR (PLC_PRG.mpx_a1_1_in_v_3 < MIN_VOLTAGE)) THEN
	ups_a1_in_v_alarm := TRUE;
ELSE
	ups_a1_in_v_alarm := FALSE;
END_IF

//Авария входного напряжения ИБПА2
IF( (PLC_PRG.mpx_a2_1_in_v_1 < MIN_VOLTAGE) OR (PLC_PRG.mpx_a2_1_in_v_2 < MIN_VOLTAGE) OR (PLC_PRG.mpx_a2_1_in_v_3 < MIN_VOLTAGE)) THEN
	ups_a2_in_v_alarm := TRUE;
ELSE
	ups_a2_in_v_alarm := FALSE;
END_IF

//------------------------------------------------------------------------------

//Авария выходного напряжения ИБПС1
IF( (PLC_PRG.mpx_s1_1_output_v_1 < MIN_VOLTAGE) OR (PLC_PRG.mpx_s1_1_output_v_2 < MIN_VOLTAGE) OR (PLC_PRG.mpx_s1_1_output_v_3 < MIN_VOLTAGE)) THEN
	ups_s1_out_v_alarm := TRUE;
ELSE
	ups_s1_out_v_alarm := FALSE;
END_IF

//Авария выходного напряжения ИБПС2
IF( (PLC_PRG.mpx_s2_1_output_v_1 < MIN_VOLTAGE) OR (PLC_PRG.mpx_s2_1_output_v_2 < MIN_VOLTAGE) OR (PLC_PRG.mpx_s2_1_output_v_3 < MIN_VOLTAGE)) THEN
	ups_s2_out_v_alarm := TRUE;
ELSE
	ups_s2_out_v_alarm := FALSE;
END_IF

//Авария выходного напряжения ИБПА1
IF( (PLC_PRG.mpx_a1_1_output_v_1 < MIN_VOLTAGE)) THEN
	ups_a1_out_v_alarm := TRUE;
ELSE
	ups_a1_out_v_alarm := FALSE;
END_IF

//Авария выходного напряжения ИБПА2
IF( (PLC_PRG.mpx_a2_1_output_v_1 < MIN_VOLTAGE)) THEN
	ups_a2_out_v_alarm := TRUE;
ELSE
	ups_a2_out_v_alarm := FALSE;
END_IF

//Авария ШАСН
IF ( (GPIO_HANDLER.IN_4 = FALSE) OR (GPIO_HANDLER.IN_5 = FALSE) ) THEN
	shasn_alarm := TRUE;
ELSE
	shasn_alarm := FALSE;
END_IF

//Авария ЩРПА
IF( (PLC_PRG.shrpa_voltage_1_line_1 < MIN_VOLTAGE) OR (PLC_PRG.shrpa_voltage_1_line_2 < MIN_VOLTAGE) OR (PLC_PRG.shrpa_voltage_1_line_3 < MIN_VOLTAGE) ) THEN
	shrpa_in_1_alarm := TRUE;	
ELSE
	shrpa_in_1_alarm := FALSE;
END_IF

IF( (PLC_PRG.shrpa_voltage_2_line_1 < MIN_VOLTAGE) OR (PLC_PRG.shrpa_voltage_2_line_2 < MIN_VOLTAGE) OR (PLC_PRG.shrpa_voltage_2_line_3 < MIN_VOLTAGE) ) THEN
	shrpa_in_2_alarm := TRUE;	
ELSE
	shrpa_in_2_alarm := FALSE;
END_IF

IF( (PLC_PRG.shrpa_voltage_3_line_1 < MIN_VOLTAGE) OR (PLC_PRG.shrpa_voltage_4_line_1 < MIN_VOLTAGE) ) THEN
	shrpa_out_alarm := TRUE;
ELSE
	shrpa_out_alarm := FALSE;
END_IF

IF ( (shrpa_in_1_alarm = TRUE) OR (shrpa_in_2_alarm = TRUE) OR (shrpa_out_alarm = TRUE) ) THEN
	schrpa_alarm := TRUE;
ELSE
	schrpa_alarm := FALSE;
END_IF

//Авария ЩРПС
IF( PLC_PRG.shrps_voltage_1_line_1 < MIN_VOLTAGE ) THEN
	shrps_in_1_alarm := TRUE;	
ELSE
	shrps_in_1_alarm := FALSE;
END_IF

IF( PLC_PRG.shrps_voltage_2_line_1 < MIN_VOLTAGE ) THEN
	shrps_in_2_alarm := TRUE;	
ELSE
	shrps_in_2_alarm := FALSE;
END_IF

IF ( (PLC_PRG.shrps_ups_bus_1 = FALSE) OR (PLC_PRG.shrps_ups_bus_2 = FALSE) ) THEN
	shrps_out_alarm_raw := TRUE;
ELSE
	shrps_out_alarm_raw := FALSE;
END_IF
Shrps_delay_timer(IN := shrps_out_alarm_raw, PT:= delay_timeout);
shrps_out_alarm :=Shrps_delay_timer.Q;

IF ( (shrps_in_1_alarm = TRUE) OR (shrps_in_2_alarm = TRUE) OR (shrps_out_alarm = TRUE) ) THEN
	schrps_alarm := TRUE;
ELSE
	schrps_alarm := FALSE;
END_IF

END_PROGRAM

// CODESYS_Control_for_Raspberry_Pi/Application/BusReinit
PROGRAM BusReinit
VAR
	BL1 : BLINK;
	BL2 : BLINK;
	BL3 : BLINK;
	BL4 : BLINK;
	BL5 : BLINK;
	BL6 : BLINK;
	BL7 : BLINK;
	BL8 : BLINK;
	BL9 : BLINK;
	BL10 : BLINK;
	BL11 : BLINK;
	BL12 : BLINK;
END_VAR

IF PLC.xError THEN 
	BL1(enable:=TRUE, timelow:=T#50MS, timehigh:=T#100MS);
	PLC.xReset:=BL1.OUT; 
	ModbusMaster.xResetComPort := TRUE;
ELSE 
	BL1(enable:=FALSE, timelow:=T#50MS, timehigh:=T#100MS);
	PLC.xReset:= FALSE;
	ModbusMaster.xResetComPort := FALSE; 
END_IF;

IF SHRPA_ICP_CON.xError THEN 
	BL2(enable:=TRUE, timelow:=T#50MS, timehigh:=T#100MS);
	SHRPA_ICP_CON.xReset:=BL2.OUT; 
	ModbusMaster.xResetComPort := TRUE;
ELSE 
	BL2(enable:=FALSE, timelow:=T#50MS, timehigh:=T#100MS);
	SHRPA_ICP_CON.xReset:= FALSE;
	ModbusMaster.xResetComPort := FALSE; 
END_IF;

IF SHRPS_ICP_CON.xError THEN 
	BL3(enable:=TRUE, timelow:=T#50MS, timehigh:=T#100MS);
	SHRPS_ICP_CON.xReset:=BL3.OUT; 
	ModbusMaster.xResetComPort := TRUE;
ELSE 
	BL3(enable:=FALSE, timelow:=T#50MS, timehigh:=T#100MS);
	SHRPS_ICP_CON.xReset:= FALSE;
	ModbusMaster.xResetComPort := FALSE; 
END_IF;

IF SHASN_ICP_CON.xError THEN 
	BL4(enable:=TRUE, timelow:=T#50MS, timehigh:=T#100MS);
	SHASN_ICP_CON.xReset:=BL4.OUT; 
	ModbusMaster.xResetComPort := TRUE;
ELSE 
	BL4(enable:=FALSE, timelow:=T#50MS, timehigh:=T#100MS);
	SHASN_ICP_CON.xReset:= FALSE;
	ModbusMaster.xResetComPort := FALSE; 
END_IF;

IF SHRPA_ELNET_1.xError THEN 
	BL5(enable:=TRUE, timelow:=T#50MS, timehigh:=T#100MS);
	SHRPA_ELNET_1.xReset:=BL5.OUT; 
	ModbusMaster.xResetComPort := TRUE;
ELSE 
	BL5(enable:=FALSE, timelow:=T#50MS, timehigh:=T#100MS);
	SHRPA_ELNET_1.xReset:= FALSE;
	ModbusMaster.xResetComPort := FALSE; 
END_IF;

IF SHRPA_ELNET_2.xError THEN 
	BL6(enable:=TRUE, timelow:=T#50MS, timehigh:=T#100MS);
	SHRPA_ELNET_2.xReset:=BL6.OUT; 
	ModbusMaster.xResetComPort := TRUE;
ELSE 
	BL6(enable:=FALSE, timelow:=T#50MS, timehigh:=T#100MS);
	SHRPA_ELNET_2.xReset:= FALSE;
	ModbusMaster.xResetComPort := FALSE; 
END_IF;

IF SHRPA_ELNET_3.xError THEN 
	BL7(enable:=TRUE, timelow:=T#50MS, timehigh:=T#100MS);
	SHRPA_ELNET_3.xReset:=BL7.OUT; 
	ModbusMaster.xResetComPort := TRUE;
ELSE 
	BL7(enable:=FALSE, timelow:=T#50MS, timehigh:=T#100MS);
	SHRPA_ELNET_3.xReset:= FALSE;
	ModbusMaster.xResetComPort := FALSE; 
END_IF;

IF SHRPA_ELNET_4.xError THEN 
	BL8(enable:=TRUE, timelow:=T#50MS, timehigh:=T#100MS);
	SHRPA_ELNET_4.xReset:=BL8.OUT; 
	ModbusMaster.xResetComPort := TRUE;
ELSE 
	BL8(enable:=FALSE, timelow:=T#50MS, timehigh:=T#100MS);
	SHRPA_ELNET_4.xReset:= FALSE;
	ModbusMaster.xResetComPort := FALSE; 
END_IF;

IF SHRPS_ELNET_1.xError THEN 
	BL9(enable:=TRUE, timelow:=T#50MS, timehigh:=T#100MS);
	SHRPS_ELNET_1.xReset:=BL9.OUT; 
	ModbusMaster.xResetComPort := TRUE;
ELSE 
	BL9(enable:=FALSE, timelow:=T#50MS, timehigh:=T#100MS);
	SHRPS_ELNET_1.xReset:= FALSE;
	ModbusMaster.xResetComPort := FALSE; 
END_IF;

IF SHRPS_ELNET_2.xError THEN 
	BL10(enable:=TRUE, timelow:=T#50MS, timehigh:=T#100MS);
	SHRPS_ELNET_2.xReset:=BL10.OUT; 
	ModbusMaster.xResetComPort := TRUE;
ELSE 
	BL10(enable:=FALSE, timelow:=T#50MS, timehigh:=T#100MS);
	SHRPS_ELNET_2.xReset:= FALSE;
	ModbusMaster.xResetComPort := FALSE; 
END_IF;

IF SHRPS_ELNET_3.xError THEN 
	BL11(enable:=TRUE, timelow:=T#50MS, timehigh:=T#100MS);
	SHRPS_ELNET_3.xReset:=BL11.OUT; 
	ModbusMaster.xResetComPort := TRUE;
ELSE 
	BL11(enable:=FALSE, timelow:=T#50MS, timehigh:=T#100MS);
	SHRPS_ELNET_3.xReset:= FALSE;
	ModbusMaster.xResetComPort := FALSE; 
END_IF;

IF SHRPS_ELNET_4.xError THEN 
	BL12(enable:=TRUE, timelow:=T#50MS, timehigh:=T#100MS);
	SHRPS_ELNET_4.xReset:=BL12.OUT; 
	ModbusMaster.xResetComPort := TRUE;
ELSE 
	BL12(enable:=FALSE, timelow:=T#50MS, timehigh:=T#100MS);
	SHRPS_ELNET_4.xReset:= FALSE;
	ModbusMaster.xResetComPort := FALSE; 
END_IF;

END_PROGRAM

// CODESYS_Control_for_Raspberry_Pi/Application/visualization/monitoring
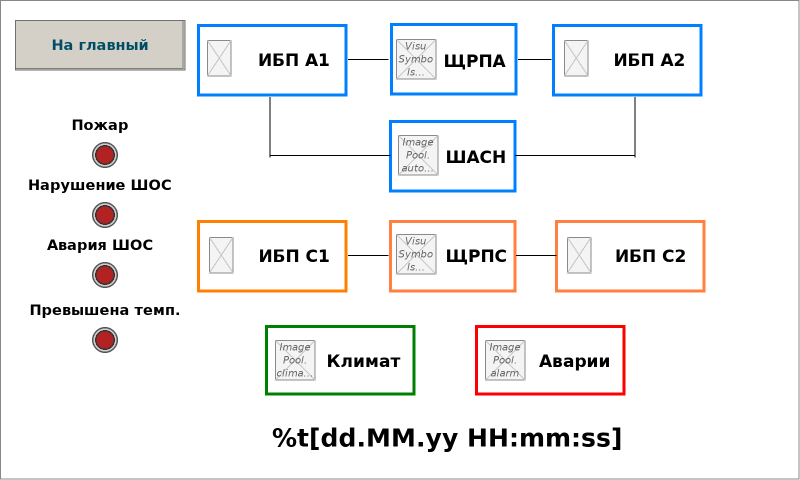
VISUALIZATION monitoring  // 800x480, background image ImagePool.bg_800
    Lamp1 (90,140 30x30), variable: GPIO_HANDLER.IN_2, style: Lamp-Lamp1-Red
    Rectangle (20,110 160x30), "Пожар"
    Lamp1 (90,200 30x30), variable: GPIO_HANDLER.IN_1, style: Lamp-Lamp1-Red
    Rectangle (20,170 160x30), "Нарушение ШОС"
    Lamp1 (90,260 30x30), variable: GPIO_HANDLER.IN_3, style: Lamp-Lamp1-Red
    Rectangle (20,230 160x30), "Авария ШОС"
    Lamp1 (90,325 30x30), variable: PLC_PRG.climate_temp_excess, style: Lamp-Lamp1-Red
    Rectangle (20,295 170x30), "Превышена темп."
    RoundedRectangle (389,220 127x72), colour toggle: AlarmChecker.schrps_alarm
    Group (396,234 118x40)
        RoundedRectangle (43,6 75x32), "ЩРПС"
            OnMouseClick:  Assign=schrps, Type=Assignment
        Image (0,0 40x40), image: VisuSymbols.Symbols.TreeDown
    Group (390,23 127x72)
        RoundedRectangle (0,0 127x72), colour toggle: AlarmChecker.schrpa_alarm
            OnMouseClick:  Assign=schrpa, Type=Assignment
        Image (6,16 40x40), image: VisuSymbols.Symbols.TreeDown
        RoundedRectangle (52,22 65x32), "ЩРПА"
            OnMouseClick:  Assign=schrpa, Type=Assignment
    Group (389,120 127x72)
        RoundedRectangle (0,0 127x72), colour toggle: AlarmChecker.shasn_alarm
            OnMouseClick:  Assign=shasn, Type=Assignment
        RoundedRectangle (48,21 78x32), "ШАСН"
            OnMouseClick:  Assign=shasn, Type=Assignment
        Image (9,15 40x40), image: ImagePool.automation-512
    Button (15,20 170x50), "На главный"
        OnMouseClick:  Assign=main, Type=Assignment
    Group (265,325 150x70)
        RoundedRectangle (0,0 150x70)
        RoundedRectangle (55,20 87x32), "Климат"
            OnMouseClick:  Assign=climate, Type=Assignment
        Image (10,15 40x40), image: ImagePool.climate
    Group (475,325 150x70)
        RoundedRectangle (0,0 150x70)
        RoundedRectangle (55,20 90x32), "Аварии"
            OnMouseClick:  Assign=alarm, Type=Assignment
        Image (10,15 40x40), image: ImagePool.alarm
    Group (197,220 150x72)
        RoundedRectangle (0,0 150x72), colour toggle: AlarmChecker.ups_s1_in_v_alarm
            OnMouseClick:  Assign=ups_s1_params, Type=Assignment
        RoundedRectangle (48,20 99x32), "ИБП С1"
            OnMouseClick:  Assign=ups_s1_params, Type=Assignment
        Image (12,17 24x36), image: ImagePool.mini_ups
    Group (555,220 150x72)
        RoundedRectangle (0,0 150x72), colour toggle: AlarmChecker.ups_s2_in_v_alarm
            OnMouseClick:  Assign=ups_s2_params, Type=Assignment
        RoundedRectangle (45,20 102x32), "ИБП С2"
            OnMouseClick:  Assign=ups_s2_params, Type=Assignment
        Image (12,17 24x36), image: ImagePool.mini_ups
    Group (197,24 150x72)
        RoundedRectangle (0,0 150x72), colour toggle: AlarmChecker.ups_a1_in_v_alarm
            OnMouseClick:  Assign=ups_a1_params, Type=Assignment
        RoundedRectangle (50,20 94x32), "ИБП А1"
            OnMouseClick:  Assign=ups_a1_params, Type=Assignment
        Image (10,16 24x36), image: ImagePool.mini_ups
    Rectangle (260,415 375x45), "%t[dd.MM.yy HH:mm:ss]"
    Group (552,24 150x72)
        RoundedRectangle (0,0 150x72), colour toggle: AlarmChecker.ups_a2_in_v_alarm
            OnMouseClick:  Assign=ups_a2_params, Type=Assignment
        RoundedRectangle (48,20 99x32), "ИБП А2"
            OnMouseClick:  Assign=ups_a2_params, Type=Assignment
        Image (12,16 24x36), image: ImagePool.mini_ups
    Line (640,130)
    Line (635,157) (635,97)
    Line (515,155) (635,155)
    Line (270,155) (390,155)
    Line (270,157) (270,97)
    Line (348,59) (388,59)
    Line (518,59) (551,59)
    Line (348,255) (388,255)
    Line (516,255) (556,255)
    hotkey  Id=481037385728, Key=KeyDown=True, KeyName=0, VisuElemId=148
    hotkey  Id=481038434304, Key=KeyName=0, VisuElemId=148
END_VISUALIZATION

// CODESYS_Control_for_Raspberry_Pi/Application/visualization/ups_s2/ups_s2_state
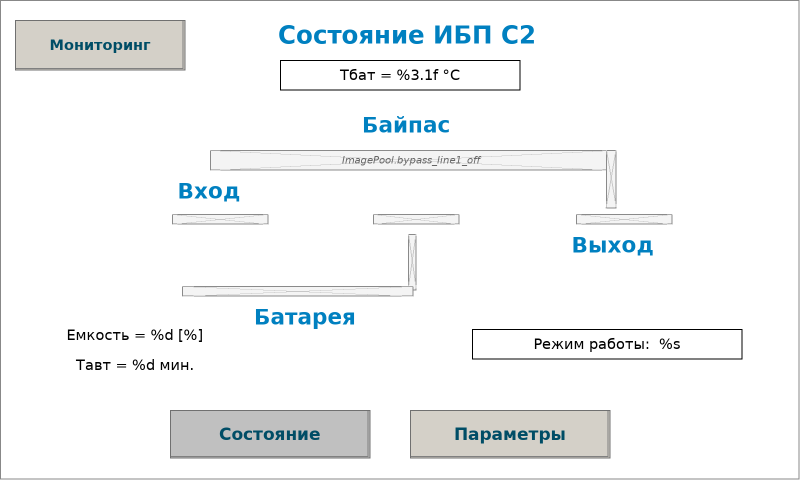
VISUALIZATION ups_s2_state  // 800x480, background image ImagePool.mpx_state_bg
    Rectangle (204,20 406x30), "Состояние ИБП С2"
    Button (410,410 200x48), "Параметры"
        OnMouseClick:  Assign=ups_s2_params, Type=Assignment
    Button (170,410 200x48), "Состояние", pressed state: PLC_PRG.var_true
    Rectangle (350,110 112x30), "Байпас"
    Rectangle (246,302 118x30), "Батарея"
    Rectangle (166,176 86x30), "Вход"
    Rectangle (560,230 106x30), "Выход"
    Rectangle (280,60 240x30), "Tбат = %3.1f °С", text variable: PLC_PRG.mpx_s2_1_temp_real
    Rectangle (30,320 210x30), "Емкость = %d [%]", text variable: PLC_PRG.mpx_s2_1_battery_capacity
    Rectangle (30,350 210x30), "Tавт = %d мин.", text variable: PLC_PRG.mpx_s2_time_m
    Image (210,150 402x20), image: ImagePool.bypass_line1_off
        p84334746: PLC_PRG.mpx_s2_1_bypass_line_state
    Image (606,150 10x58), image: ImagePool.bypass_arrow_off
        p84334746: PLC_PRG.mpx_s2_1_bypass_arrow_state
    Image (576,214 96x10), image: ImagePool.arrow_off
        p84334746: PLC_PRG.mpx_s2_1_output_state
    Image (172,214 96x10), image: ImagePool.arrow_off
        p84334746: PLC_PRG.mpx_s2_1_input_state
    Image (408,234 8x56), image: ImagePool.battery_arrow_off
        p84334746: PLC_PRG.mpx_s2_1_battery_arrow_state
    Image (182,286 231x10), image: ImagePool.battery_line_off
        p84334746: PLC_PRG.mpx_s2_1_battery_line_state
    Button (15,20 170x50), "Мониторинг"
        OnMouseClick:  Assign=monitoring, Type=Assignment
    Rectangle (372,212 85x14)
    Image (373,214 86x10), image: ImagePool.arrow_off
        p84334746: PLC_PRG.mpx_s2_1_arrow_state
    Rectangle (472,329 270x30), "Режим работы: %s", text variable: PLC_PRG.mpx_s2_state_string
    hotkey  Id=481037385728, Key=KeyDown=True, KeyName=0, VisuElemId=38
    hotkey  Id=481038434304, Key=KeyName=0, VisuElemId=38
END_VISUALIZATION

